# B&R Automation Studio project ABC_Pltzr
Automation Studio 4.2.2.134


## Configuration PPC70_Ver1

### Hardware
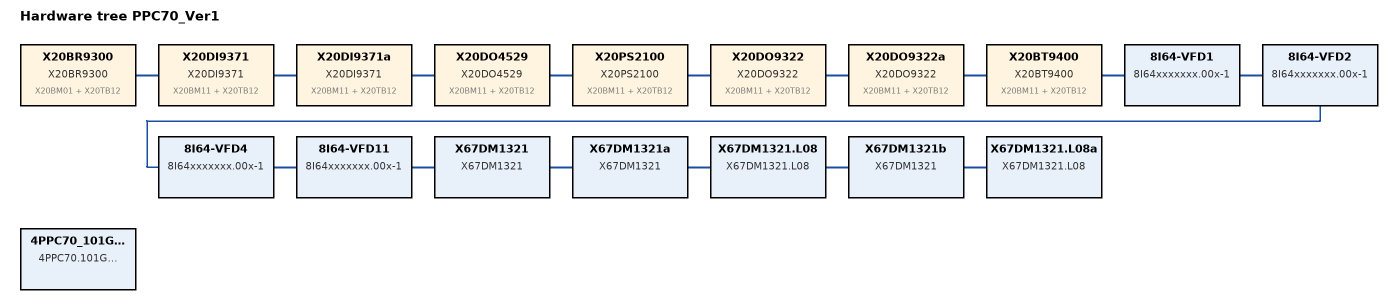
```
4PPC70_101G_20F005 : 4PPC70.101G-20F005 v1.1.0.0
  Connector IF1:
    ActivatePowerlink = 0
  Connector IF2:
    ActivateDevice = 1
    Mode = Manual
    InternetAddress = 192.168.1.100
    SubnetMask = 255.255.255.0
    InaNodeNumber = 1
    Vnc1
    VncVcObjectName1 = WSVGA
    VncKeyMappingFile1 = VC\PS2-Keyboard.dis
    VncAuthentication1 = 1
    VncPasswordViewOnly1 = v
    VncPasswordViewControl1 = eric
  Simulation = 1
  PermanentPvSize = 1000
  RemanentGlobalPvSize = 25000
  VolatileGlobalPvSize = 200000
  EnableUsbRemoteInstall = 1
  TimerDeviceType = SWIOTIMER
  Cyclic1Duration = 4000
  Cyclic1Tolerance = 4000
  Cyclic2Duration = 20000
  Cyclic2Tolerance = 20000
  Cyclic3Duration = 50000
  Cyclic3Tolerance = 50000
  Cyclic4Duration = 100000
  Cyclic4Tolerance = 100000
  Cyclic5Duration = 200000
  Cyclic5Tolerance = 200000
  Cyclic6Duration = 500000
  Cyclic6Tolerance = 500000
  Cyclic7Duration = 1000000
  Cyclic7Tolerance = 1000000
  Cyclic8Duration = 10000
  Cyclic8Tolerance = 30000000
  FtpUser1
  FtpUsername1 = abc
  FtpUserPassword1 = veVz20Da1KUF2Vww53L6omFNdzfk8lHY0HjcrjfOb/w=  // abc123
  FtpUserSalt1 = pyAcjG26
  FTPPath1 = 5
  FTPAccessRight1 = 0
  VcObjectName = WSVGA
  KeyMappingFile = VC\4PPC70_101G_20F005.dis
8I64-VFD1 : 8I64xxxxxxx.00x-1 v1.3.8.1  [X2X1 -> X20BT9400.X2X1]
  FunctionModel = Standard
  Supervision = off
  enableIOLR = off
  enableDigitalOutput = off
  DigitalOutputMode01 = actionDO
  ACC = 1
  DEC = 1
  LSP = 10
  HSP = 600
  ITH = 28
  BFR = 1
  UNS = 460
  FRS = 600
  NCR = 28
  NSP = 1750
  COS = 80
  DO = 9
  BRA = 0
  BLC = 64
  BRT = 15
  BEN = 0
  BET = 15
8I64-VFD11 : 8I64xxxxxxx.00x-1 v1.3.8.1  [X2X1 -> 8I64-VFD4.X2X2]
  FunctionModel = Standard
  Supervision = off
  enableIOLR = off
  enableDigitalOutput = off
  HSP = 600
  FTD = 600
  BFR = 1
  UNS = 460
  FRS = 600
  NCR = 15
  NSP = 1750
  COS = 80
8I64-VFD2 : 8I64xxxxxxx.00x-1 v1.3.8.1  [X2X1 -> 8I64-VFD1.X2X2]
  FunctionModel = Standard
  Supervision = off
  enableIOLR = off
  enableDigitalOutput = off
  DigitalOutputMode01 = actionDO
  DownloadParameters = yes
  ACC = 1
  DEC = 1
  BFR = 1
  UNS = 460
  FRS = 600
  NCR = 13
  NSP = 1750
  DO = 9
  BRA = 0
  BLC = 64
  BRT = 5
  BEN = 0
  BET = 5
8I64-VFD4 : 8I64xxxxxxx.00x-1 v1.3.8.1  [X2X1 -> 8I64-VFD2.X2X2]
  FunctionModel = Standard
  Supervision = off
  enableIOLR = off
  enableDigitalOutput = off
  DigitalOutputMode01 = actionDO
  DownloadParameters = yes
  ACC = 1
  DEC = 1
  HSP = 600
  ITH = 13
  FTD = 600
  BFR = 1
  UNS = 460
  FRS = 600
  NCR = 13
  NSP = 1750
  COS = 80
  DO = 9
  BRA = 0
  BLC = 64
  BRT = 5
  BEN = 0
  BET = 5
X20BM01 : X20BM01 v1.0.0.1
X20BM11 : X20BM11 v1.0.0.0  [X2X1 -> X20BM01.X2X2]
X20BM11a : X20BM11 v1.0.0.0  [X2X1 -> X20BM11.X2X2]
X20BM11b : X20BM11 v1.0.0.0  [X2X1 -> X20BM11a.X2X2]
X20BM11c : X20BM11 v1.0.0.0  [X2X1 -> X20BM11b.X2X2]
X20BM11d : X20BM11 v1.0.0.0  [X2X1 -> X20BM11c.X2X2]
X20BM11e : X20BM11 v1.0.0.0  [X2X1 -> X20BM11f.X2X2]
X20BM11f : X20BM11 v1.0.0.0  [X2X1 -> X20BM11d.X2X2]
X20BR9300 : X20BR9300 v1.0.2.6  [SS1 -> X20TB12.SS; SL -> X20BM01.SL1; X2X1 -> 4PPC70_101G_20F005.IF5]
  Supervision = off
X20BT9400 : X20BT9400 v1.0.1.3  [SS1 -> X20TB12f.SS; SL -> X20BM11e.SL1]
  Supervision = off
X20DI9371 : X20DI9371 v1.0.1.2  [SS1 -> X20TB12a.SS; SL -> X20BM11.SL1]
  Supervision = off
X20DI9371a : X20DI9371 v1.0.1.2  [SS1 -> X20TB12b.SS; SL -> X20BM11a.SL1]
  Supervision = off
  InputFilter = 100
X20DO4529 : X20DO4529 v1.0.1.2  [SS1 -> X20TB12c.SS; SL -> X20BM11b.SL1]
  Supervision = off
X20DO9322 : X20DO9322 v1.0.2.2  [SS1 -> X20TB12e.SS; SL -> X20BM11d.SL1]
  Supervision = off
X20DO9322a : X20DO9322 v1.0.2.2  [SS1 -> X20TB12g.SS; SL -> X20BM11f.SL1]
  Supervision = off
X20PS2100 : X20PS2100 v1.0.3.0  [SS1 -> X20TB12d.SS; SL -> X20BM11c.SL1]
  Supervision = off
X20TB12 : X20TB12 v1.0.0.0
X20TB12a : X20TB12 v1.0.0.0
X20TB12b : X20TB12 v1.0.0.0
X20TB12c : X20TB12 v1.0.0.0
X20TB12d : X20TB12 v1.0.0.0
X20TB12e : X20TB12 v1.0.0.0
X20TB12f : X20TB12 v1.0.0.0
X20TB12g : X20TB12 v1.0.0.0
X67DM1321 : X67DM1321 v1.1.1.0  [X2X1 -> 8I64-VFD11.X2X2]
  Supervision = off
X67DM1321.L08 : X67DM1321.L08 v1.1.2.0  [X2X1 -> X67DM1321a.X2X2]
  Supervision = off
  Direction01 = output
  Direction02 = output
  Direction03 = output
  Direction04 = output
  Direction05 = output
  Direction06 = output
  Direction07 = output
  Direction08 = output
  Direction09 = output
  Direction10 = output
  Direction11 = output
  Direction12 = output
X67DM1321.L08a : X67DM1321.L08 v1.1.2.0  [X2X1 -> X67DM1321b.X2X2]
  Supervision = off
  Direction08 = output
  Direction09 = output
X67DM1321a : X67DM1321 v1.1.1.0  [X2X1 -> X67DM1321.X2X2]
  Supervision = off
  Direction01 = output
  Direction02 = output
  Direction03 = output
  Direction04 = output
X67DM1321b : X67DM1321 v1.1.1.0  [X2X1 -> X67DM1321.L08.X2X2]
  Supervision = off
```

## Configuration testsim

CPU , AutomationRuntime D4.22, Build 4.1.2, Vc V4.22.0

### Config_1.mprecipexml - PLC1/mapp/Config_1.mprecipexml
```
Element gMpLinkMpRecipeXml (Type=mprecipexml)
```

## Logical view

Binary libraries used (declarations not repeated): AsBrStr, AsMath, AsTCP, AsUSB, Ethernet

### Program Logical/appConfigAndRecipes/appCfgRec

#### appCfgRec.c
```c
/********************************************************************
 * COPYRIGHT -- piedmont
 ********************************************************************
 * Program: cfgFS
 * File: cfgFS.c
 * Author: admin
 * Created: Jan 20, 2014
 ********************************************************************
 * Implementation of program cfgFS
 ********************************************************************/

#include <bur/plctypes.h>

#ifdef _DEFAULT_INCLUDES
 #include <AsDefault.h>
#endif

/**
 Simple logging
 Log goes to an array of PV strings > see _LOCAL STRING log[][] variable below
 Log output is visible via Automation Studio watch window
 Example of a log statement used within the code is:
 DBG("This is log example. %d ", value1);
 To complety disable logging from this source file, change next line to: #if 0
*/
#if 1
#include <../../paiComponents/bglib/bgPVLogger3.c>
#define LOG_ENTRY_COUNT 30	//max number of log entries
#define LOG_ENTRY_LENGTH  200//max length of individual log message. Longer msg are truncated
_LOCAL STRING log[LOG_ENTRY_COUNT][LOG_ENTRY_LENGTH]; //log output visible from Automation Studio!
//static bgPVLogger_typ lgr;	//PV logger object
#else
#define DBG(format, args...) ;
#define DBGINIT(args...) ;
#endif

//Support for PV serialization/deserialization
#include "../../paiComponents/bglib/bgPVSerialize.h"
#include "../appCfgRecDefault.h"
#include "../../paiComponents/paiFileService/paiPVSerDesMgr.h"
#include "../../paiComponents/paiFileService/paiFSInterface.h"
#include "../../paiComponents/paiFileService/paiFS/paiFile.h"
#include "../../paiComponents/Libraries/sprintf2/sprintf2.h"

/*
###############################################################################
PV-s
###############################################################################
*/

/*
###############################################################################
Functions
###############################################################################
*/

static void fileSetCfgFilePath(char* pCfgFilePath)
{
//Example:
//Output: pRecFilePath = "ABC/appcfg.txt"
	sprintf2(pCfgFilePath, "%s/%s", APP_DIR_NAME, APP_FILENAME_CFG);
}

/*
###############################################################################
Remanent Memory Handling
- remanent (REM) memory is battery backed SRAM
- unlike files, it has a fast, pointer based access
- in this application, it is used as a first level of storage, as follows

  working memory (DRAM) data
- valid only while CPU powered
- working memory holds all PV-s and application strucutres

Remanent memory (SRAM battery backed)
- power fail safe (only WARM restart! COLD restart deletes remanent memory)
- selected structures (eg. machine confiuration, current recipe) are copied into this area as a first level backup
- fast backup via simple memcpy

Files (CF disk)
- power fail safe and permanent
- backup requires use of FileIO access (slower, more complex)

This application combines use of the above mentioned memories.

IMPORTANT:
The REMMEM support was added before realizing that most CPU-s support only tiny (eg. 32 bytes) REM Memory areas.
As a result, the REM memory support is not really working as intended. The intended REMMEM PV-s are stored as
regular PV-s which means that these values are not preserved during power cycle.
###############################################################################
*/

static void defineFileNames()
{
	//file that holds machine configuration
	//Example: cfgFilename = "Data/appcfg.txt"
	fileSetCfgFilePath(cfgFilename);

}

/*
###############################################################################
Init, Cyclic, Exit
###############################################################################
*/
void paiPVSerDesMgrConfigure();

void _INIT appCfgRecInit( void )
{
	/* TODO: Add code here */
	DBGINIT(lgr, log, LOG_ENTRY_COUNT, LOG_ENTRY_LENGTH);

	//Define file names used for storign PV-s in this application
	defineFileNames();			//define file names used in this application

	//Configure paiSerDesMgr
	paiPVSerDesMgrConfigure();

	//TODO: gRecipe
	brsstrcpy((UDINT)gRecipe.info.name, (UDINT)"ABC");
}

void _CYCLIC appCfgRecCyclic( void )
{

	//paiFS callback execution cyclic service
	//This service executes File IO related callbacks in the context of this task
	paiFSExeCallbackCyclic(&paiFS);

	//paiSerDesMgr cyclic
	paiPVSerDesMgrCyclic(&gPVSerDesMgr);
}
//EOF
```

### notes.txt
```
9/21/2016
=========
(ProjectDate:='09/21/2016',ProjectVersion:='1.00.2',ASVersion:='AS 4.2.4',ProjectAbout:='Palletizer72',ProjectInfo:='24025',ProjectComments:='n/a')

-------- Forwarded Message --------
Subject: 	Duckhorn Wine
Date: 	Fri, 9 Sep 2016 13:25:31 +0000
From: 	David Emminger <demminger@abcpackaging.com>
To: 	Goran Bjelcevic <gbjelcevic@piedmontautomation.com>
CC: 	Eric Dederichs <edederichs@abcpackaging.com>, Greg Phelps <gphelps@piedmontautomation.com>, Kraig Downey <kdowney@abcpackaging.com>, Brittany Leslie <bleslie@abcpackaging.com>

Good morning Goran,
Duckhorn has requested a minor change to the machine HMI programming which is:

They want the fault screen to remain displayed and not automatically close when a fault is cleared. They want to manually navigate away from the fault screen.

Unhide the mute button

Change the maintenance access password to 4858418

- a logic to automaticaly switch away from the alarm screen when all alarms are cleared is removed.
Change: file: appHmiLogic.c, line: 1491
- changed the maint access password to 4858418
Change: file: paiUser.c, line: 105
- changed hide logic for safety curtains 'mute' button. Now, the button will be shown even for users that are not logged in.
Change: ladder: palletdischarge Rung: 13

5/2/2016
=======
-rectified 'no pallet reset' after executing 'Complete Pallet' manual request
-changed logic for stopping the infeed CV; instead of stopping when staging stops, the infeed CV now stops only when staging is stopped AND case is present at EE2
-changed logic for elevator when exiting pallet; instead of going to top of the pallet, now the elevator goes to the top (max elevator position)
-fixed issue with entering a case command in the layer desinger
-added support for 6th blade
-changed manual operation of the blade stops from time delayed to quick (no time delay)

4/18/2016
==========
DONE-EE2 / EE8 stop the machine row jam/incorrect count
DONE-stage at EE4
DONE-stats timer only in auto mode
-vfd fault indication in the alarm text
DONE-prevent changing counts in automatic
DONE-in automatic can't go to manual screen (put finish product button eslewhere)
-full pallet out should zero the layers
DONE ALARM INCORRECT COUNT
DONE HIDE ZERO BUTTON WHEN in AUTO
VFD BRA = OFF for VFD5 and VFD52

4/15/2016
=========
DONE: Button: load appConfig from file
VFD errors show in the alarm!
Stats counters
Case count
Pallete count
Pallete / hour
Case / min
DONE: Blade stop drawing support
DONE: Move blade stop timers to recipe
Staging cv support
Usb programming
File copy to/from to usb
Factory defaults
Retainer bar early feature
Pallet discharge interlock
Remove unused code, pages, etc
Add stop / resume to ssm.
Add single step support to ssm.

4/14/12016
=========
DONE-moved all timers to recipe
DONE-added pallet exit button (manual mode only)
DONE-added pallet finish button (auto mode only, to finish pallet and discharge)
-

4/13/2015
==========
- zero button visibility check logic (it can cause havoc is pressed when not allowed)
DONE- pallet done (in auto mode, compeltes the pallete and exits it)
 vs. run pallet out (in manual mode, exits the palette) > buttons needed
STOP BUTTON - shall stop and any time, then resume from there
PART- debounce timers for all PE-s (EE2, EE4, EE8) > recipe
DONE - product/recipe dependant settings (i.e. timers, etc)
DONE- delay front squearing action using a delay timer
DONE- pallet takeaway timer; the time required for a discharge PE to clear before the pallet are moved to discharge cv forward
- EE8 get the code for it
DONE- row forming VFD speeds and acc, table speed, acc/decl, discrage cv-s > all VDD-s shall be part of the recipe
DONE - defending fault shall be shown as the alarm!! (not low air pressure)
DONE - drop down LF key to jump to screen MANUAL
DONE - the delay time for row push shall be respected after restart following an e-stop on the last case for the row (if the e-stop tiggered just before the last estop made the row, the continue will immedialtly push the
row wo. waiting)
- Connect Alarm Ack button to the Clear VFD Fault input

3/24/2015
==========
-add alarm for elevator stop block
-add light curtain functionlity - fault and mute
-chain slack alarm recovery from stop block
-add message block stops are down

3/23/2015
=========
-added support for new HW config:
PPC70_JOB24025
-this configuration is according to the ABC JOB24025
-no palletizer dispneser is used. Instead, the pallets are build directly onto the mesh converyer
-the HW changes include:
-added 2 VFD-s VFD52 (row pusher ext) and VFD12 (pallet discharge CV)
-dropped VFD4 (row pusher) and reassinged it as VFD5 (infeed rollers)

3/22/2016
==========
-revisit and rectify recipe handling to have only a single file per recipe (i.e. layer files included in the recipe file)
-DONE-reshuffle recipe screens (i.e. recipe select, recipe create, layer create, layer view, etc)
DONE-add support for multiple blade stops
DONE-add support for pallet dispenser
-add support for infeed conveyer location (left/right) to be reflected on the configuration screen
DONE-rectify issue with the VFD-s at startup (i.e. reboot shall not be required due to incorrect configuration)
-revisti all hmi screens
-test interruptions, e-stops and power outages
-allow elevator jog when table not at grouping (recovery mode!)
-add new alarms
-pattern layer changes require reload of the pattern program to init the structures!!!

2/15/2016
==========
-revisit and rectify recipe handling to have only a single file per recipe (i.e. layer files included in the recipe file)
-reshuffle recipe screens (i.e. recipe select, recipe create, layer create, layer view, etc)
-add support for multiple blade stops
-add support for pallet dispenser
-add support for infeed conveyer location (left/right) to be reflected on the configuration screen
-rectify issue with the VFD-s at startup (i.e. reboot shall not be required due to incorrect configuration)
-revisti all hmi screens
-test interruptions, e-stops and power outages
-allow elevator jog when table not at grouping (recovery mode!)

9/10/2015
========-
-DONEadd blade stops
-DONEadd turner
-DONEestop handling
-DONEacc/dec on all drives
-DONEadd configurable number of layers

9/9/2015
=========
-add messages about zerooing machine
-add message about machine ready
-add message when auto-cycle active
-start/auto drycycle sequence

9/4/2013
========
-add number of E-Stops as an option into mach configuration
-add number of DS-s as an option into mach configuration
-add discharge light curtain to the safety logic
-remove AlwaysOnBit and TestBitx from the program when done

-add manual elevator moves to table position (use two speeds)

7/22/2015
-io
-control strructures
-alarms
-recipes
-control logic
-hmi

Subsystems:
===========
Motors ON/OFF:
-retainer bar
-row/grouping rollers
-product infeed cv
-pallet infeed chains
-pallet dispense elevator

Inverters:
-elevator
-transfer table
-row pusher
-palletizing roller cv

Machine Modes:
==============
Service (Air=NO, all motors = OFF)
Manual - HandMode (Air=YES, all motors = ON, NOT in automatic mode, manual actions)
Auto - MachineRunningAuto (automatic cycle)
DryCycle (automatic, dry cycle)
Demo (automatic, demo cycle)

Original LADDERS:
-main
-screen
-IO
-dispenser
-inserter
-bladestop1...bladestop6
-squaring
-prodset
-patterns
-picture
-caserun
-stdturner
-turntable
-servoturn
-drycycle
```

### Global.typ
```iecst
(********************************************************************
 * COPYRIGHT -- HP
 ********************************************************************
 * File: Global.typ
 * Author: goran
 * Created: January 23, 2013
 ********************************************************************
 * Global data types of project YieldPlus
 ********************************************************************)

TYPE
	applicationGlobal_enums :
		(
		APP_HWMODULE_IDXLAST := 19, (*Number of  X20 HW modules*)
		APP_CFG_BLADESTOP_MAXIDX := 5, (*Max number of blade stops*)
		APP_VFD_IDXLAST := 12 (*Max number of VFD-s*)
		);
END_TYPE
```

### Global.var
```iecst
(********************************************************************
 * COPYRIGHT -- HP
 ********************************************************************
 * File: Global.var
 * Author: goran
 * Created: January 23, 2013
 ********************************************************************
 * Global variables of project YieldPlus
 ********************************************************************)
VAR
	gProjectInfo : {REDUND_UNREPLICABLE} paiProjectInfo_typ := (ProjectDate:='09/21/2016',ProjectVersion:='1.00.2',ASVersion:='AS 4.2.4',ProjectAbout:='Palletizer72',ProjectInfo:='24025',ProjectComments:='n/a');
END_VAR
VAR RETAIN
	gREMMEMPrefix : UDINT;
	gREMMEMPostfix : UDINT;
END_VAR
```

- AlarmPopUp.fninfo (not shown)

- Arial9px.fninfo (not shown)

- Arial9pxBold.fninfo (not shown)

- Html_SDM_0.fninfo (not shown)

- Pads.fninfo (not shown)

- EditPad.tpr (not shown)

- MpNavigationPad_ver.tpr (not shown)

### brsystem.var
```iecst
(********************************************************************
 * COPYRIGHT (C) BERNECKER + RAINER, AUSTRIA, A-5142 EGGELSBERG
 ********************************************************************
 * Library: BrSystem
 * File: BrSystem.var
 * Created: 11.11.2003
 ********************************************************************
 * Constants of library BrSystem
 ********************************************************************)
VAR CONSTANT
	brSYSCONF_SET_NON_VOLATILE	: BOOL	:= TRUE;	(*set permanent value*)
	brERR_INVALID_PARAMETER	: UINT	:= 27251;		(*invalid parameter transferred*)
	brSYSCONF_SET_VOLATILE	: BOOL	:= FALSE;		(*set non-permanent value*)
	INIT_REASON_WARMSTART	: SINT	:= 1;			(*warm restart boot information*)
	INIT_REASON_COLDSTART	: SINT	:= 2;			(*cold restart boot information*)
	brERR_INVALID_DEVICE	: UINT	:= 27250;		(*battery monitoring*)
	brAUTOMATION_RUNTIME	: USINT	:= 4;			(*series recognition*)
	TARGET_LITTLE_ENDIAN	: USINT	:= 1;			(*formatSpec*)
	INIT_REASON_DOWNLOAD	: SINT	:= 3;			(*download boot information*)
	INIT_REASON_UNKNOWN	: SINT	:= -1;				(*unknown boot information*)
	brBATTERY_MISSING	: USINT	:= 3;				(*battery monitoring*)
	TARGET_BIG_ENDIAN	: USINT	:= 2;				(*formatSpec*)
	brBATTERY_NOTEST	: USINT	:= 2;				(*battery monitoring*)
	brSYSTEM_MODULE	: USINT	:= 2;					(*usage recognition*)
	brPLUGIN_MODULE	: USINT	:= 10;					(*usage recognition*)
	brLOGICSCANNER	: USINT	:= 3;					(*series recognition*)
	brBATTERY_LOW	: USINT	:= 0;					(*battery monitoring*)
	brPOWERPANEL	: USINT	:= 5;					(*series recognition*)
	brBATTERY_OK	: USINT	:= 1;					(*battery monitoring*)
	brREMOTE_IO	: USINT	:= 4;						(*usage recognition*)
	brNO_FAMILY	: USINT	:= 255;						(*series recognition*)
	brETHER_IO	: USINT	:= 6;						(*usage recognition*)
	brPRODUCT	: USINT	:= 0;						(*usage recognition*)
	brBASE_IO	: USINT	:= 3;						(*usage recognition*)
	brCAN_IO	: USINT	:= 5;						(*usage recognition*)
	brACOPOS	: USINT	:= 7;						(*usage recognition*)
	brUSRRAM	: UDINT	:= 1;						(*USRRAM memory type*)
	brSYSROM	: UDINT	:= 2;						(*SYSROM memory type*)
	brUSRROM	: UDINT	:= 3;						(*USRROM memory type*)
	brPANEL	: USINT	:= 6;							(*series recognition*)
	brADDON	: USINT	:= 7;							(*series recognition*)
	brC300	: USINT	:= 8;							(*series recognition*)
	brC200	: USINT	:= 9;							(*series recognition*)
	br2010	: USINT	:= 0;							(*series recognition*)
	br2005	: USINT	:= 1;							(*series recognition*)
	br2003	: USINT	:= 2;							(*series recognition*)
	brDRAM	: UDINT	:= 0;							(*DRAM memory type*)
	brKEY	: USINT	:= 8;							(*usage recognition*)
	brCPU	: USINT	:= 1;							(*usage recognition*)
	brPP	: USINT	:= 255;							(*usage recognition*)
	brX2X	: USINT	:= 10;							(*series recognition*)
END_VAR
```

### dvframe.var
```iecst
(********************************************************************
 * COPYRIGHT (C) BERNECKER + RAINER, AUSTRIA, A-5142 EGGELSBERG
 ********************************************************************
 * Library:    DVFrame
 * File:            DVFrame.var
 * Created:         11.11.2003
 ********************************************************************
 * Constants of library DVFrame
 ********************************************************************)
VAR CONSTANT
	frmERR_IOCTL_NOTSUPPORTED	: UINT	:= 8257;	(*command not supported by driver (hardware)*)
	frmERR_DEVICEDESCRIPTION	: UINT	:= 8252;	(*device not found*)
	frmERR_FUB_ENABLE_FALSE	: UINT	:= 65534;
	frmERR_TRANSMITOVERRUN	: UINT	:= 8078;		(*send buffer waiting queue full*)
	frmERR_MODEDESCRIPTION	: UINT	:= 8253;		(*syntax error in mode parameter string, or mode parameter not supported by the specified device*)
	frmERR_IOCTL_NOTVALID	: UINT	:= 8073;		(*invalid I/O control code*)
	frmERR_INVALIDBUFFER	: UINT	:= 8072;		(*invalid buffer rejected*)
	ARG_EVSEND_TASKIDENT	: UDINT	:= 14;
	ARG_EVSEND_TASKEVENT	: UDINT	:= 18;
	frmERR_NORESOURCES	: UINT	:= 8258;			(*required resource not available (memory, OS object, etc.)*)
	frmERR_INPUTERROR	: UINT	:= 8079;			(*frame buffer with defective character*)
	frmERR_NOTOPENED	: UINT	:= 8251;			(*device not open*)
	MISC_RECEIVE_ALL	: UDINT	:= 2;
	frmERR_PA_DB_SB	: UINT	:= 8256;				(*/PA, /DB, /SB must always be specified together*)
	frmERR_NOBUFFER	: UINT	:= 8071;				(*no buffer available in the send buffer manager*)
	ARG_TXPVPOLLADR	: UDINT	:= 17;
	frmERR_NOINPUT	: UINT	:= 60;					(*no message received*)
	frmERR_MAXOPEN	: UINT	:= 8254;				(*too many devices opened at once*)
	ARG_PVPOLLADR	: UDINT	:= 15;
	frmERR_OK	: UINT	:= 0;
	ARG_MISC	: UDINT	:= 16;
	ARG_BAUD	: UDINT	:= 0;
END_VAR
```

- vssver.scc (binary file, 48 bytes)
### MpFile.typ
```iecst
TYPE
	MpFileManagerUIItemType : 	STRUCT
		Name : STRING[255]; (*Filename / Folder name*)
		Size : UDINT; (*File size [bytes]*)
		LastModified : DATE_AND_TIME; (*Date when this file/folder was last modified*)
		ItemType : MpFileManagerUIItemTypeEnum; (*File type (.csv, .jpg, etc.)*)
		IsSelected : BOOL; (*Indicates that a file/folder is selected*)
		IsFolder : BOOL; (*Indicates that the element is a folder*)
	END_STRUCT;
	MpFileManagerUIItemTypeEnum :
		(
		mpFILE_ITEM_TYPE_NONE := 0, (*No type defined*)
		mpFILE_ITEM_TYPE_FOLDER := 1, (*Indicates that the element is a folder*)
		mpFILE_ITEM_TYPE_FILE := 2, (*Indicates that the element is a file*)
		mpFILE_ITEM_TYPE_TXT := 3, (*Indicates that the element is a text file*)
		mpFILE_ITEM_TYPE_HTML := 4, (*Indicates that the element is an HTML file*)
		mpFILE_ITEM_TYPE_DOC := 5, (*Indicates that the element is a Word file (.doc) *)
		mpFILE_ITEM_TYPE_XLS := 6, (*Indicates that the element is an Excel file (.xls)*)
		mpFILE_ITEM_TYPE_XML := 7, (*Indicates that the element is an XML file (.xml)*)
		mpFILE_ITEM_TYPE_CSV := 8, (*Indicates that the element is an CSV file (.csv)*)
		mpFILE_ITEM_TYPE_JPG := 9, (*Indicates that the element is an image file (.jpg)*)
		mpFILE_ITEM_TYPE_BMP := 10, (*Indicates that the element is an image file (.bmp)*)
		mpFILE_ITEM_TYPE_USER1 := 89, (*Indicates that the element is an user predefined type 1*)
		mpFILE_ITEM_TYPE_USER2 := 90, (*Indicates that the element is an user predefined type 2*)
		mpFILE_ITEM_TYPE_USER3 := 91, (*Indicates that the element is an user predefined type 3*)
		mpFILE_ITEM_TYPE_USER4 := 92, (*Indicates that the element is an user predefined type 4*)
		mpFILE_ITEM_TYPE_USER5 := 93, (*Indicates that the element is an user predefined type 5*)
		mpFILE_ITEM_TYPE_USER6 := 94, (*Indicates that the element is an user predefined type 6*)
		mpFILE_ITEM_TYPE_USER7 := 95, (*Indicates that the element is an user predefined type 7*)
		mpFILE_ITEM_TYPE_USER8 := 96, (*Indicates that the element is an user predefined type 8*)
		mpFILE_ITEM_TYPE_USER9 := 97, (*Indicates that the element is an user predefined type 9*)
		mpFILE_ITEM_TYPE_USER10 := 98, (*Indicates that the element is an user predefined type 10*)
		mpFILE_ITEM_TYPE_UNKNOWN := 99 (*Indicates that the file type is unknown*)
		);
	MpFileManagerUISortOrderEnum :
		(
		mpFILE_SORT_BY_NAME_ASC := 0, (*Sorts in ascending (alphabetic) order*)
		mpFILE_SORT_BY_NAME_DESC := 1, (*Sorts in descending (alphabetic) order*)
		mpFILE_SORT_BY_SIZE_ASC := 2, (*Sorts in ascending order by file size*)
		mpFILE_SORT_BY_SIZE_DES := 3, (*Sorts in descending order by file size*)
		mpFILE_SORT_BY_MOD_TIME_ASC := 4, (*Sorts in ascending order by date last modified*)
		mpFILE_SORT_BY_MOD_TIME_DESC := 5 (*Sorts in descending order by date last modified*)
		);
	MpFileManagerUIMessageEnum :
		(
		mpFILE_MSG_OK := 0, (*Dialog box for requesting confirmation of input*)
		mpFILE_MSG_CONFIRM_DELETE := 1, (*Dialog box for requesting confirmation of deletion*)
		mpFILE_MSG_CONFIRM_OVERWRITE := 2, (*Dialog box for requesting confirmation of overwriting*)
		mpFILE_MSG_BUSY := 3 (*Dialog box for requesting confirmation of busy UI*)
		);
	MpFileDiagType : 	STRUCT
		StatusID : MpFileStatusIDType; (*StatusID diagnostic structure*)
	END_STRUCT;
	MpFileStatusIDType : 	STRUCT
		ID : MpFileErrorEnum; (*Error code for mapp component*)
		Severity : MpComSeveritiesEnum; (*Describes the type of information supplied by the status ID (success, information, warning, error)*)
		Code : UINT; (*Code for the status ID. This error number can be used to search for additional information in the help system.*)
	END_STRUCT;
	MpFileInfoType : 	STRUCT
		Diag : MpFileDiagType; (*Diagnostic structure for the status ID*)
	END_STRUCT;
	MpFileManagerUIStatusEnum :
		(
		mpFILE_UI_STATUS_IDLE := 0, (*Indicates that no process is currently active*)
		mpFILE_UI_STATUS_REFRESH := 1, (*Updating elements*)
		mpFILE_UI_STATUS_CHANGE_PAGE := 2, (*Page change active*)
		mpFILE_UI_STATUS_CHANGE_DIR := 3, (*Folder change active*)
		mpFILE_UI_STATUS_CHANGE_DEVICE := 4, (*File Device Change active*)
		mpFILE_UI_STATUS_CREATE := 5, (*Creating a file/folder active*)
		mpFILE_UI_STATUS_RENAME := 6, (*Renaming a file/folder active*)
		mpFILE_UI_STATUS_DELETE := 7, (*Deleting a file/folder active*)
		mpFILE_UI_STATUS_COPY := 8, (*Copying a file/folder active*)
		mpFILE_UI_STATUS_CUT := 9, (*Cutting a file/folder active*)
		mpFILE_UI_STATUS_PASTE := 10, (*Pasting a file/folder active*)
		mpFILE_UI_STATUS_SORT := 11, (*Sorting files/folders in specified sort order*)
		mpFILE_UI_STATUS_ERROR := 99 (*The last operation generated an error*)
		);
	MpFileManagerUISetupType : 	STRUCT
		FileListSize : UINT := 10; (*Number of files to be displayed on one page of the list in the HMI application*)
		FileListScrollWindow : USINT := 1; (*Determines how many entries from the list are displayed in advance when scrolling up and down*)
	END_STRUCT;
	MpFileManagerUIConnectType : 	STRUCT
		Status : MpFileManagerUIStatusEnum; (*Current operation*)
		DeviceList : MpFileManagerUIDeviceListType; (*List of data storage media (file devices) accessible by the file manager*)
		File : MpFileManagerUIFileType; (*Contains the file list as well as additional information about files,folders and possible commands*)
		MessageBox : MpFileManagerUIMessageBoxType; (*Controls dialog boxes*)
		DefaultLayerStatus : UINT; (*Status DP for the default layer of the visu page where the file manager is being displayed*)
	END_STRUCT;
	MpFileManagerUIMessageBoxType : 	STRUCT
		LayerStatus : UINT; (*Visibility of the dialog box*)
		Type : MpFileManagerUIMessageEnum; (*Type of dialog box*)
		ErrorNumber : UINT; (*Current error number to be displayed*)
		Confirm : BOOL; (*Confirms the operation*)
		Cancel : BOOL; (*Cancels the operation*)
	END_STRUCT;
	MpFileManagerUIPathInfoType : 	STRUCT
		CurrentDir : STRING[255]; (*Current folder name*)
		FileCount : UDINT; (*Number of files in the current folder*)
		FolderCount : UDINT; (*Number of subfolders in the current folder*)
	END_STRUCT;
	MpFileManagerUIFileType : 	STRUCT
		List : MpFileManagerUIFileListType; (*List of all folders and files under the current path, as well as the navigation of the list*)
		Filter : STRING[255]; (*Filter used to sort the files*) (* *) (*#CMD#OPT#;*)
		SortOrder : MpFileManagerUISortOrderEnum; (*Responsible for the order of files in the list*)
		Refresh : BOOL; (*Updates the file list in the current folder*)
		PathInfo : MpFileManagerUIPathInfoType; (*Information about the current path*)
		EnterFolder : BOOL; (*Navigates one folder down*)
		FolderUp : BOOL; (*Navigates one folder up*)
		MultiSelect : BOOL; (*Allows the selection of multiple elements at the same time*)
		Delete : BOOL; (*Deletes a file or folder*)
		Copy : BOOL; (*Copying a file/folder*)
		Cut : BOOL; (*Cuts a file or folder*)
		Paste : BOOL; (*Pastes a file or folder*)
		NewName : STRING[255]; (*The new name of a file or folder when using the "Rename" or "CreateFolder" command*)
		Rename : BOOL; (*Renames a file or folder*)
		CreateFolder : BOOL; (*Creates a folder*)
	END_STRUCT;
	MpFileManagerUIFileListType : 	STRUCT
		Items : ARRAY[0..49]OF MpFileManagerUIItemType; (*List of all files and folders under the current path*)
		PageUp : BOOL; (*Jumps to the start of the current page and then scrolls up one page at a time*)
		StepUp : BOOL; (*Selects the previous entry in the list*)
		PageDown : BOOL; (*Jumps to the end of the current page and then scrolls down one page at a time*)
		StepDown : BOOL; (*Selects the next entry in the list*)
		RangeStart : REAL; (*Shows a bar indicating which part of the list is currently being displayed-Start [%]*)
		RangeEnd : REAL; (*Shows a bar indicating which part of the list is currently being displayed-End [%]*)
	END_STRUCT;
	MpFileManagerUIDeviceListType : 	STRUCT
		DeviceNames : ARRAY[0..9]OF STRING[50]; (*List of all available data storage media*)
		SelectedIndex : UINT; (*Index of the entry currently selected in the list*)
	END_STRUCT;
END_TYPE
```

- vssver.scc (binary file, 48 bytes)
- Program Logical/MachineControl/animation (IEC) (no source held here)

### Program Logical/MachineControl/appHmi

#### appHmiLogic.c
```c
/********************************************************************
 * COPYRIGHT -- pai
 ********************************************************************
 * Program: hmilogic
 * File: hmilogic.c
 * Author: goran
 * Created: August 28, 2013
 ********************************************************************
 * Implementation of program hmilogic
 ********************************************************************/

#include <bur/plctypes.h>

#ifdef _DEFAULT_INCLUDES
	#include <AsDefault.h>
#endif

#include "../../paiComponents/paiHmi/paiHmiParamList.h"
#include "../../paiComponents/paiHmi/paiHmiPageChange.h"
#include "../../paiComponents/paiHmi/paiHmiAlert.h"
#include "../../paiComponents/bglib/bgBitUtilities.h"

/*
###############################################################################
Utilities
###############################################################################
*/

/**
Screen ID-s must match AutomationStudio's  VisualComponents Page Numbers!!!!!
NOTE: not all screen must have logic support written in this file! Actually,
less logic here and using more VC features is a prefered approach to
implement VC HMI apps.
*/
enum{
	SID_Init = 0,
	SID_Main = 10,
	SID_Main_Monitor = 11,
	SID_Settings_System = 60,
	SID_Settings_Timers = 61,
	SID_Settings_VFDs = 62,
	SID_Settings_Options = 63,
	SID_Settings_MachCfg = 65,
	SID_Recipe_LayerDesign = 44,
	SID_Recipe_LayerPreview = 41,
	SID_Recipe_PalletSelect = 46,
	SID_Recipe_PalletConfig = 45,
	SID_Recipe_PalletTimers = 47,
	SID_Recipe_PalletVFDs = 48,
	SID_Diag_Alarms = 81,
	SID_System_Files = 103,
	SID_Manual = 82,
	SID_Manual2 = 87,

	SID_MAX  /*always last!!!*/
}APPSCREENIDS;

/**
Application specific HMI dialogs must be unique. Always to in pair (accept,reject, etc)
*/
enum{
	DLG_Ok = 10,
	DLG_Cancel,
	DLG_DeleteL1FilenameOK = 20,
	DLG_DeleteL1FilenameCancel,
	DLG_SaveAppConfigOK = 30,
	DLG_SaveAppConfigCancel,
	DLG_SavePalletRecipeOK = 40,
	DLG_SavePalletRecipeCancel,

}APPHMIDIALOGIDS;

/*
###############################################################################
Parameter view/edit tables
###############################################################################
*/

/*
###############################################################################
Parameter view/edit tables
###############################################################################
*/
static void hmiTableRecipeTimers()
{
	//configApp_typ* pAppCfg = &gConfigApp;
	palleteCfgSettings_typ* pAppCfg = &gPallete.palCfg.palSettings;

	//	DINT decFormat_None = -2; //no dec places
	//	DINT decFormat_0 = -1;    //1 dec place
	DINT decFormat_00 = 0;    //default (2) dec places as set in the control
	//	DINT decFormat_000 = 1;    //3 dec places

	//scaling
	//y=kx+n where: y=HMI value, x=PLC value
	REAL k_factor = 1.0;
	REAL n_factor = 0.0;
	//	UINT valtypeUDINT = 0;//UDINT
	UINT valtypeREAL = 1;//REAL

	hmiParamListTableEntryFirst(&gHmiParamTable, "Pallet Timers");

//#if 0
	hmiParamListTableAddEntryNext(&gHmiParamTable,
		(UDINT)&pAppCfg->timers.dlyTableLayerRdyToElevMove , "TableReadyToElevatorMove",
		1.0, 0.1, 5.0,
		decFormat_00, k_factor, n_factor, valtypeREAL, "Delay time from Table Layer Ready to Elevator Move [sec].");

	hmiParamListTableAddEntryNext(&gHmiParamTable,
		(UDINT)&pAppCfg->timers.dlyTableAtPalleteToRetBar , "DelayRetainerBarMoveDown",
		1.0, 0.1, 5.0,
		decFormat_00, k_factor, n_factor, valtypeREAL, "Delay time from Table at Pallet to Retainer Bar move down to Squaring [sec].");

	hmiParamListTableAddEntryNext(&gHmiParamTable,
		(UDINT)&pAppCfg->timers.onDlyPRRetBarDown , "DelayRetainerBarIsDown",
		0.05, 0.00, 1.0,
		decFormat_00, k_factor, n_factor, valtypeREAL, "On delay for Retainer Bar Down Prox sensor [sec]. Higher value > layer edge gets positioned deeper inside the pallete.");

	hmiParamListTableAddEntryNext(&gHmiParamTable,
		(UDINT)&pAppCfg->timers.onDlyEEPallete , "onDelayEE1Pallet",
		0.05, 0.00, 1.0,
		decFormat_00, k_factor, n_factor, valtypeREAL, "On delay for Pallet Sensor EE1[sec]. Longer delay results in table getting closer to the pallete when dropping a layer. DANGER: Setting this time too long may cause mechanical colision!");

	hmiParamListTableAddEntryNext(&gHmiParamTable,
		(UDINT)&pAppCfg->timers.offDlyEEPallete , "offDelayEE1Pallet",
		0.05, 0.00, 3.0,
		decFormat_00, k_factor, n_factor, valtypeREAL, "Off delay for Pallet Sensor EE1[sec].");

	hmiParamListTableAddEntryNext(&gHmiParamTable,
		(UDINT)&pAppCfg->timers.onDlyPalleteDischargeEE16 , "onDelayPalleteDischargeEE16",
		0.05, 0.00, 3.0,
		decFormat_00, k_factor, n_factor, valtypeREAL, "On delay for Pallet Discharge Sensor EE16[sec]. Longer delay results in pallete getting futher on the discharge CV. DANGER: Setting this time too long may cause pallete tip over!");

	hmiParamListTableAddEntryNext(&gHmiParamTable,
		(UDINT)&pAppCfg->timers.onTmCaseTurner , "onTimeCaseTurner",
		1.0, 0.1, 5.0,
		decFormat_00, k_factor, n_factor, valtypeREAL, "On Time for case turner[sec].");

	hmiParamListTableAddEntryNext(&gHmiParamTable,
		(UDINT)&pAppCfg->timers.dlyRowDoneToRowPush , "DelayForRowDoneToRowPush",
		1.0, 0.1, 5.0,
		decFormat_00, k_factor, n_factor, valtypeREAL, "Delay time from row forming conmplete signal to push the row to the table [sec].");

	hmiParamListTableAddEntryNext(&gHmiParamTable,
		(UDINT)&pAppCfg->timers.dlyLastCaseToRowCVStop , "DelayLastCaseToRowConvStop",
		1.0, 0.1, 5.0,
		decFormat_00, k_factor, n_factor, valtypeREAL, "Delay from the moment the last case for a row passes by EE4 until a row forming CV is stopped[sec].");

	hmiParamListTableAddEntryNext(&gHmiParamTable,
		(UDINT)&pAppCfg->timers.dlyPusherAtElevatorToRetract , "DelayPusherAtElevatorReturnToHome",
		1.0, 0.1, 5.0,
		decFormat_00, k_factor, n_factor, valtypeREAL, "Delay from the moment row pusher gets to the elevator before a reverse motion is started to retract row pusher back to home[sec].");

	hmiParamListTableAddEntryNext(&gHmiParamTable,
		(UDINT)&pAppCfg->timers.dlyTableAtPalleteToRetBar , "DelayTableFwdToRetainerBarDown",
		1.0, 0.0, 5.0,
		decFormat_00, k_factor, n_factor, valtypeREAL, "Delay from a moment the table starts moving towards the pallet top and before a retainter bar starts moving down[sec]. NOTE: Setting this value too short may cause a collision.");

	hmiParamListTableAddEntryNext(&gHmiParamTable,
		(UDINT)&pAppCfg->timers.onDlyTableToGrouping , "DelayTableToGrouping",
		0.0, 0.0, 2.0,
		decFormat_00, k_factor, n_factor, valtypeREAL, "Delay from a moment the layer is dropped onto the top of the pallet and before table starts moving towards the grouping[sec].");

	hmiParamListTableAddEntryNext(&gHmiParamTable,
		(UDINT)&pAppCfg->timers.JamAlarmTmAtInfeedEE2 , "JamAlarmTimeAtCaseInfeedEE2",
		4.0, 1.0, 20.0,
		decFormat_00, k_factor, n_factor, valtypeREAL, "Maximum time allowed to block the EE2 Case Infeed PE before a jam alarm is generated [sec].");

	hmiParamListTableAddEntryNext(&gHmiParamTable,
		(UDINT)&pAppCfg->timers.JamAlarmTmAtRowToLongEE8 , "JamAlarmTimeAtRowToLongEE8",
		4.0, 1.0, 20.0,
		decFormat_00, k_factor, n_factor, valtypeREAL, "Maximum time allowed to block the EE8 Row Too Long PE before an alarm is generated [sec].");

	hmiParamListTableAddEntryNext(&gHmiParamTable,
		(UDINT)&pAppCfg->timers.JamAlarmTmRowForming , "JamAlarmTimeAtRowForming",
		4.0, 1.0, 20.0,
		decFormat_00, k_factor, n_factor, valtypeREAL, "Maximum time allowed for a case to travel between EE2 (Case Infeed PE) and EE8 (Row Too Long PE) before an alarm is generated [sec].");

	hmiParamListTableAddEntryNext(&gHmiParamTable,
		(UDINT)&pAppCfg->timers.infeedCVIdleTime , "InfeedCVIdleTime",
		30.0, 10.0, 600.0,
		decFormat_00, k_factor, n_factor, valtypeREAL, "Maximum idle time for infeed CV-s before they get turned off[sec].");

	hmiParamListTableAddEntryNext(&gHmiParamTable,
		(UDINT)&pAppCfg->timers.palletExitAlarmTm , "PalletExitAlarmTime",
		15.0, 5.0, 60.0,
		decFormat_00, k_factor, n_factor, valtypeREAL, "Maximum time allowed for a pallet to exit the machine (i.e. activate EE16) [sec].");
//#endif

	hmiParamListTableAddEntryNext(&gHmiParamTable,
		(UDINT)&pAppCfg->timers.EE2OnDebounce , "EE2OnDebounce",
		0.0, 0.0, 0.5,
		decFormat_00, k_factor, n_factor, valtypeREAL, "EE2 (Infeed) On debounce time[sec].");

	hmiParamListTableAddEntryNext(&gHmiParamTable,
		(UDINT)&pAppCfg->timers.EE2OfDebounce , "EE2OffDebounce",
		0.0, 0.0, 0.5,
		decFormat_00, k_factor, n_factor, valtypeREAL, "EE2 (Infeed) Off debounce time[sec].");

	hmiParamListTableAddEntryNext(&gHmiParamTable,
		(UDINT)&pAppCfg->timers.EE4OnDebounce , "EE4OnDebounce",
		0.0, 0.0, 0.5,
		decFormat_00, k_factor, n_factor, valtypeREAL, "EE4 (Stage CV PE) On debounce time[sec].");

	hmiParamListTableAddEntryNext(&gHmiParamTable,
		(UDINT)&pAppCfg->timers.EE4OfDebounce , "EE4OffDebounce",
		0.0, 0.0, 0.5,
		decFormat_00, k_factor, n_factor, valtypeREAL, "EE4 (Stage CV PE) Off debounce time[sec].");

	hmiParamListTableAddEntryNext(&gHmiParamTable,
		(UDINT)&pAppCfg->timers.EE8OnDebounce , "EE8OnDebounce",
		0.0, 0.0, 0.5,
		decFormat_00, k_factor, n_factor, valtypeREAL, "EE8 (Row To Long) On debounce time[sec].");

	hmiParamListTableAddEntryNext(&gHmiParamTable,
		(UDINT)&pAppCfg->timers.EE8OfDebounce , "EE8OffDebounce",
		0.0, 0.0, 0.5,
		decFormat_00, k_factor, n_factor, valtypeREAL, "EE8 (Row To Long) Off debounce time[sec].");

	hmiParamListTableAddEntryNext(&gHmiParamTable,
		(UDINT)&pAppCfg->timers.EE16OfDebounce , "EE16OffDebounce",
		5.0, 0.0, 60.0,
		decFormat_00, k_factor, n_factor, valtypeREAL, "EE16 (Pallete Discharge Sensor) Off debounce time[sec]. Longer time prevents to quick exiting of a pallete from the staging CV to discharge CV after EE16 gets unblocked.");

	hmiParamListTableAddEntryNext(&gHmiParamTable,
		(UDINT)&pAppCfg->timers.onDlyFrontSquaring , "FrontSquaringOnDelay",
		0.0, 0.0, 3.0,
		decFormat_00, k_factor, n_factor, valtypeREAL, "Front Squaring On Delay[sec]. Allows for a delayed action of the front squaring bar to prevent product pushing.");

	if(gConfigApp.system.bladeStopCount >= 1){
		hmiParamListTableAddEntryNext(&gHmiParamTable,
			(UDINT)&pAppCfg->timers.bladeStopOnDly1 , "Blade1TurnOnDelay",
			1.0, 0.0, 10.0,
			decFormat_00, k_factor, n_factor, valtypeREAL, "Blade 1 turn-on delay. Delayed turn-on when executing pattern program is required so that the blade does not block an incorrect case [sec].");
	}

	if(gConfigApp.system.bladeStopCount >= 2){
		hmiParamListTableAddEntryNext(&gHmiParamTable,
			(UDINT)&pAppCfg->timers.bladeStopOnDly2 , "Blade2TurnOnDelay",
			2.0, 0.0, 10.0,
			decFormat_00, k_factor, n_factor, valtypeREAL, "Blade 2 turn-on delay. Delayed turn-on when executing pattern program is required so that the blade does not block an incorrect case [sec]");
	}

	if(gConfigApp.system.bladeStopCount >= 3){
		hmiParamListTableAddEntryNext(&gHmiParamTable,
			(UDINT)&pAppCfg->timers.bladeStopOnDly3 , "Blade3TurnOnDelay",
			3.0, 0.0, 10.0,
			decFormat_00, k_factor, n_factor, valtypeREAL, "Blade 3 turn-on delay. Delayed turn-on when executing pattern program is required so that the blade does not block an incorrect case [sec]");
	}

	if(gConfigApp.system.bladeStopCount >= 4){
		hmiParamListTableAddEntryNext(&gHmiParamTable,
			(UDINT)&pAppCfg->timers.bladeStopOnDly4 , "Blade4TurnOnDelay",
			4.0, 0.0, 10.0,
			decFormat_00, k_factor, n_factor, valtypeREAL, "Blade 4 turn-on delay. Delayed turn-on when executing pattern program is required so that the blade does not block an incorrect case [sec]");
	}

	if(gConfigApp.system.bladeStopCount >= 5){
		hmiParamListTableAddEntryNext(&gHmiParamTable,
			(UDINT)&pAppCfg->timers.bladeStopOnDly5 , "Blade5TurnOnDelay",
			5.0, 0.0, 10.0,
			decFormat_00, k_factor, n_factor, valtypeREAL, "Blade 5 turn-on delay. Delayed turn-on when executing pattern program is required so that the blade does not block an incorrect case [sec]");
	}

	hmiParamListTableEntryLast(&gHmiParamTable);

}

static void hmiTableOptions()
{
	configApp_typ* pAppCfg = &gConfigApp;

	DINT decFormat_None = -2; //no dec places
//	DINT decFormat_0 = -1;    //1 dec place
	DINT decFormat_00 = 0;    //default (2) dec places as set in the control
//	DINT decFormat_000 = 1;    //3 dec places

	//scaling
	//y=kx+n where: y=HMI value, x=PLC value
	REAL k_factor = 1.0;
	REAL n_factor = 0.0;
	UINT valtypeUDINT = 0;//UDINT
	UINT valtypeREAL = 1;//REAL

	hmiParamListTableEntryFirst(&gHmiParamTable, "Options");

	hmiParamListTableAddEntryNext(&gHmiParamTable,
		(UDINT)&pAppCfg->options.dryCycleCaseCount, "DryCycleCaseCount",
		5.0, 1.0, 5.0,
		decFormat_None, k_factor, n_factor, valtypeUDINT, "Number of cases per row during DryCycle.");

	hmiParamListTableAddEntryNext(&gHmiParamTable,
		(UDINT)&pAppCfg->options.dryCycleRowCount, "DryCycleRowCount",
		4.0, 1.0, 4.0,
		decFormat_None, k_factor, n_factor, valtypeUDINT, "Number of rows per layer during DryCycle.");

	hmiParamListTableAddEntryNext(&gHmiParamTable,
		(UDINT)&pAppCfg->options.dryCycleLayerCount, "DryCycleLayerCount",
		3.0, 1.0, 6.0,
		decFormat_None, k_factor, n_factor, valtypeUDINT, "Number of layers on the pallet during DryCycle.");

	hmiParamListTableAddEntryNext(&gHmiParamTable,
		(UDINT)&pAppCfg->options.tmDryCycleElevatorUp, "DryCycleElevatorUp Time",
		3.0, 1.0, 5.0,
		decFormat_00, k_factor, n_factor, valtypeREAL, "DryCycle simulation timer for simulating layers [sec].");

	hmiParamListTableAddEntryNext(&gHmiParamTable,
		(UDINT)&pAppCfg->options.tmDryCycleCaseTime , "DryCycleCase Time",
		2.0, 1.0, 5.0,
		decFormat_00, k_factor, n_factor, valtypeREAL, "DryCycle simulation time for simulating loading a single case [sec].");

	hmiParamListTableAddEntryNext(&gHmiParamTable,
		(UDINT)&pAppCfg->options.tmDryCycleLayerZeroOffset , "DryCycleLayer0Offset",
		2.0, 1.0, 5.0,
		decFormat_00, k_factor, n_factor, valtypeREAL, "DryCycle layer 0 offset time. Alows elevator position control for the layer 0. [sec].");

	hmiParamListTableAddEntryNext(&gHmiParamTable,
		(UDINT)&pAppCfg->options.dryCycleLayerDonePause , "DryCyclePause",
		0.0, 0.0, 1.0,
		decFormat_None, k_factor, n_factor, valtypeUDINT, "0-continues DryCycle operation, 1-pause after layer completion during DryCycle.");

	hmiParamListTableEntryLast(&gHmiParamTable);

}

static void hmiTableRecipeVFDs()
{
	//configApp_typ* pAppCfg = &gConfigApp;
	palleteCfgSettings_typ* pAppCfg = &gPallete.palCfg.palSettings;

	DINT decFormat_None = -2; //no dec places
	//DINT decFormat_0 = -1;    //1 dec place
	//DINT decFormat_00 = 0;    //default (2) dec places as set in the control
	//	DINT decFormat_000 = 1;    //3 dec places

	//scaling
	//y=kx+n where: y=HMI value, x=PLC value
	REAL k_factor = 1.0;
	REAL n_factor = 0.0;
	UINT valtypeUDINT = 0;//UDINT
	//	UINT valtypeREAL = 1;//REAL

	hmiParamListTableEntryFirst(&gHmiParamTable, "Pallet VFD Settings");

	hmiParamListTableAddEntryNext(&gHmiParamTable,
		(UDINT)&pAppCfg->vfd[1].velocity_rpm, "VelocityVFD1",
		300.0, 0.0, 2700.0,
		decFormat_None, k_factor, n_factor, valtypeUDINT, "VFD1(Elevator) Velocity [rpm]");

	hmiParamListTableAddEntryNext(&gHmiParamTable,
		(UDINT)&pAppCfg->vfd[1].velocitySlow_rpm, "VelocityVFD1Slow",
		150.0, 0.0, 2700.0,
		decFormat_None, k_factor, n_factor, valtypeUDINT, "VFD1(Elevator) Slow Velocity. Used when approaching home position [rpm]");

	hmiParamListTableAddEntryNext(&gHmiParamTable,
		(UDINT)&pAppCfg->vfd[2].velocity_rpm, "VelocityVFD2",
		300.0, 0.0, 2700.0,
		decFormat_None, k_factor, n_factor, valtypeUDINT, "VFD2(Table) Velocity [rpm]");
#if 0
	hmiParamListTableAddEntryNext(&gHmiParamTable,
		(UDINT)&pAppCfg->vfd[4].velocity_rpm, "VelocityVFD4",
		300.0, 0.0, 2700.0,
		decFormat_None, k_factor, n_factor, valtypeUDINT, "VFD4(Row Pusher) Velocity [rpm]");
#endif

	hmiParamListTableAddEntryNext(&gHmiParamTable,
		(UDINT)&pAppCfg->vfd[5].velocity_rpm, "VelocityVFD5",
		300.0, 0.0, 2700.0,
		decFormat_None, k_factor, n_factor, valtypeUDINT, "VFD5 Row Forming Rollers Velocity [rpm]");

	hmiParamListTableAddEntryNext(&gHmiParamTable,
		(UDINT)&pAppCfg->vfd[6].velocity_rpm, "VelocityVFD52",
		300.0, 0.0, 2700.0,
		decFormat_None, k_factor, n_factor, valtypeUDINT, "VFD52 Row Forming Rollers 2 Velocity [rpm]");

	hmiParamListTableAddEntryNext(&gHmiParamTable,
		(UDINT)&pAppCfg->vfd[11].velocity_rpm, "VelocityVFD11",
		300.0, 0.0, 2700.0,
		decFormat_None, k_factor, n_factor, valtypeUDINT, "VFD11 (Pallet Forming Mesh CV) Velocity [rpm]");

	hmiParamListTableAddEntryNext(&gHmiParamTable,
		(UDINT)&pAppCfg->vfd[12].velocity_rpm, "VelocityVFD12",
		300.0, 0.0, 2700.0,
		decFormat_None, k_factor, n_factor, valtypeUDINT, "VFD12(Pallet Discharge Mesh CV) Velocity [rpm]");

	//Acceleration
	hmiParamListTableAddEntryNext(&gHmiParamTable,
		(UDINT)&pAppCfg->vfd[1].acc, "AccelVFD1",
		1.0, 1.0, 10.0,
		decFormat_None, k_factor, n_factor, valtypeUDINT, "VFD1(Elevator) Acceleration [0.1 sec]");

	hmiParamListTableAddEntryNext(&gHmiParamTable,
		(UDINT)&pAppCfg->vfd[2].acc, "AccelVFD2",
		1.0, 1.0, 20.0,
		decFormat_None, k_factor, n_factor, valtypeUDINT, "VFD2(Table) Acceleration [0.1 sec]");

	hmiParamListTableAddEntryNext(&gHmiParamTable,
		(UDINT)&pAppCfg->vfd[5].acc, "AccelVFD5",
		1.0, 1.0, 20.0,
		decFormat_None, k_factor, n_factor, valtypeUDINT, "VFD5(Row Forming Rollers) Acceleration [0.1 sec]");

	hmiParamListTableAddEntryNext(&gHmiParamTable,
		(UDINT)&pAppCfg->vfd[6].acc, "AccelVFD52",
		1.0, 1.0, 20.0,
		decFormat_None, k_factor, n_factor, valtypeUDINT, "VFD52(Row Forming Rollers 2) Acceleration [0.1 sec]");

	hmiParamListTableAddEntryNext(&gHmiParamTable,
		(UDINT)&pAppCfg->vfd[11].acc, "AccelVFD11",
		1.0, 1.0, 200.0,
		decFormat_None, k_factor, n_factor, valtypeUDINT, "VFD11(Forming Mesh CV) Acceleration [0.1 sec]");

	hmiParamListTableAddEntryNext(&gHmiParamTable,
		(UDINT)&pAppCfg->vfd[12].acc, "AccelVFD12",
		1.0, 1.0, 200.0,
		decFormat_None, k_factor, n_factor, valtypeUDINT, "VFD12(Exit Mesh CV) Acceleration [0.1 sec]");

	//Deceleration
	hmiParamListTableAddEntryNext(&gHmiParamTable,
		(UDINT)&pAppCfg->vfd[1].dec, "DecelVFD1",
		1.0, 0.0, 10.0,
		decFormat_None, k_factor, n_factor, valtypeUDINT, "VFD1(Elevator) Deceleration [0.1 sec]");

	hmiParamListTableAddEntryNext(&gHmiParamTable,
		(UDINT)&pAppCfg->vfd[2].dec, "DecelVFD2",
		1.0, 0.0, 20.0,
		decFormat_None, k_factor, n_factor, valtypeUDINT, "VFD2(Table) Deceleration [0.1 sec]");

	hmiParamListTableAddEntryNext(&gHmiParamTable,
		(UDINT)&pAppCfg->vfd[5].dec, "DecelVFD5",
		1.0, 0.0, 20.0,
		decFormat_None, k_factor, n_factor, valtypeUDINT, "VFD5(Row Forming Rollers) Deceleration [0.1 sec]");

	hmiParamListTableAddEntryNext(&gHmiParamTable,
		(UDINT)&pAppCfg->vfd[6].dec, "DecelVFD52",
		1.0, 0.0, 20.0,
		decFormat_None, k_factor, n_factor, valtypeUDINT, "VFD52(Row Forming Rollers 2) Deceleration [0.1 sec]");

	hmiParamListTableAddEntryNext(&gHmiParamTable,
		(UDINT)&pAppCfg->vfd[11].dec, "DecelVFD11",
		1.0, 0.0, 200.0,
		decFormat_None, k_factor, n_factor, valtypeUDINT, "VFD11(Forming Mesh CV) Deceleration [0.1 sec]");

	hmiParamListTableAddEntryNext(&gHmiParamTable,
		(UDINT)&pAppCfg->vfd[12].dec, "DecelVFD12",
		1.0, 0.0, 200.0,
		decFormat_None, k_factor, n_factor, valtypeUDINT, "VFD12(Exit Mesh CV) Deceleration [0.1 sec]");

	hmiParamListTableEntryLast(&gHmiParamTable);

}

static void hmiTableMachCfg()
{
	configApp_typ* pAppCfg = &gConfigApp;

	DINT decFormat_None = -2; //no dec places
	DINT decFormat_0 = -1;    //1 dec place
	//DINT decFormat_00 = 0;    //default (2) dec places as set in the control
//	DINT decFormat_000 = 1;    //3 dec places

	//scaling
	//y=kx+n where: y=HMI value, x=PLC value
	REAL k_factor = 1.0;
	REAL n_factor = 0.0;
	UINT valtypeUDINT = 0;//UDINT
	UINT valtypeREAL = 1;//REAL

	hmiParamListTableEntryFirst(&gHmiParamTable, "Mechanical Properties");

	hmiParamListTableAddEntryNext(&gHmiParamTable,
		(UDINT)&pAppCfg->options.optTearSheetEquiped, "TierSheetPresent",
		0.0, 0.0, 1.0,
		decFormat_None, k_factor, n_factor, valtypeUDINT, "1-Machine is equiped with a tier sheet inserting assembly.");

	hmiParamListTableAddEntryNext(&gHmiParamTable,
		(UDINT)&pAppCfg->options.optOption1Equiped, "Option1Present",
		0.0, 0.0, 1.0,
		decFormat_None, k_factor, n_factor, valtypeUDINT, "1-Machine is equipped with Option1 assembly.");

	hmiParamListTableAddEntryNext(&gHmiParamTable,
		(UDINT)&pAppCfg->options.palletDispenserOption, "PalletDispenserOption",
		0.0, 0.0, 1.0,
		decFormat_None, k_factor, n_factor, valtypeUDINT, "0-Pallet Dispenser Is NOT Present/NOT Equipped; 1-Pallet Dispenser is present/equipped.");

	hmiParamListTableAddEntryNext(&gHmiParamTable,
		(UDINT)&pAppCfg->options.frontSquaringOption, "FrontSquaringOption",
		0.0, 0.0, 1.0,
		decFormat_None, k_factor, n_factor, valtypeUDINT, "0-Front Squaring assembly Is NOT Present/NOT Equipped; 1-Front Squaring assembly is present/equipped.");

	hmiParamListTableAddEntryNext(&gHmiParamTable,
		(UDINT)&pAppCfg->system.boxInfeedSide, "InfeedLeftOrRight",
		0.0, 0.0, 1.0,
		decFormat_None, k_factor, n_factor, valtypeUDINT, "0-Box infeed Right to Left. 1-Box infeed Left to Right. Point of reference: person standing in front of the row pusher assembly looking towards the layer forming table.");

	hmiParamListTableAddEntryNext(&gHmiParamTable,
		(UDINT)&pAppCfg->system.simulationMode , "SimulationMode",
		0.0, 0.0, 1.0,
		decFormat_None, k_factor, n_factor, valtypeUDINT, "Simulation Mode. 0-OFF, 1-ON (Testing only!)");

	hmiParamListTableAddEntryNext(&gHmiParamTable,
		(UDINT)&pAppCfg->system.bladeStopCount, "NumberOfBladeStops",
		0.0, 0.0, 6.0,
		decFormat_None, k_factor, n_factor, valtypeUDINT, "Total number of blade stops on the machine.");

	hmiParamListTableAddEntryNext(&gHmiParamTable,
		(UDINT)&pAppCfg->system.bladeStopDistance[0] , "BladeStop1Distance",
		10.0, 0.0, 100.0,
		decFormat_0, k_factor, n_factor, valtypeREAL, "Distance/position of the blade stop 1 [inch]. Blade 1 is ALWAYS the blade closest to the infeed/incoming side of the row forming CV.");

	hmiParamListTableAddEntryNext(&gHmiParamTable,
		(UDINT)&pAppCfg->system.bladeStopDistance[1] , "BladeStop2Distance",
		12.0, 0.0, 100.0,
		decFormat_0, k_factor, n_factor, valtypeREAL, "Distance/position of the blade stop 2 [inch]");

	hmiParamListTableAddEntryNext(&gHmiParamTable,
		(UDINT)&pAppCfg->system.bladeStopDistance[2] , "BladeStop3Distance",
		14.0, 0.0, 100.0,
		decFormat_0, k_factor, n_factor, valtypeREAL, "Distance/position of the blade stop 3 [inch]");

	hmiParamListTableAddEntryNext(&gHmiParamTable,
		(UDINT)&pAppCfg->system.bladeStopDistance[3] , "BladeStop4Distance",
		16.0, 0.0, 100.0,
		decFormat_0, k_factor, n_factor, valtypeREAL, "Distance/position of the blade stop 4 [inch]");

	hmiParamListTableAddEntryNext(&gHmiParamTable,
		(UDINT)&pAppCfg->system.bladeStopDistance[4] , "BladeStop5Distance",
		18.0, 0.0, 100.0,
		decFormat_0, k_factor, n_factor, valtypeREAL, "Distance/position of the blade stop 5 [inch]");

	hmiParamListTableEntryLast(&gHmiParamTable);
}

//control visibility of the INPUT field (layer) for the parametar edit/view table
static void loginLevelParameterEditControl(UDINT minRights, UDINT minLevel)
{
	//controlling the locking of the editing form
	//(i.e. to lock > visibility set to 0 (visible) as the flag is used for a touch area over the inputs
	gHmiParamTable.selValueFormVisible = ((gPaiUserMgr.currentGroup.AccessRights[0] >= minRights) && (gPaiUserMgr.currentGroup.Level >= minLevel)) ? 1 : 0;
}

/*
###############################################################################
HMI screen handling logic
###############################################################################
*/
void screenHandlers(paiHmiTemplate_typ* pHmi)
{
	//Page specific init logic
	if(pHmi->prv.pageInit){
		//control visibility of the parametar input form

		//screen init event
		//define screen name
		switch(pHmi->runtime.pageCurrent){
			case SID_Settings_Timers:
			break;
			case SID_Settings_MachCfg:
				loginLevelParameterEditControl(mpUSER_ACCESS_FULL, 100); //only manufacturer
				hmiTableMachCfg();
			break;
			case SID_Settings_Options:
				loginLevelParameterEditControl(mpUSER_ACCESS_FULL, 100); //only manufacturer
				hmiTableOptions();
				break;
			case SID_Settings_VFDs:
				break;
			case SID_Recipe_PalletTimers:
				loginLevelParameterEditControl(mpUSER_ACCESS_FULL, 20); //normaly, supervisor is allowed to change data
				hmiTableRecipeTimers();
				break;
			case SID_Recipe_PalletVFDs:
				loginLevelParameterEditControl(mpUSER_ACCESS_FULL, 20); //normaly, supervisor is allowed to change data
				hmiTableRecipeVFDs();
				break;
			case SID_Main_Monitor:
			case SID_Recipe_PalletSelect:
			case SID_Recipe_PalletConfig:
			case SID_System_Files:
			case SID_Recipe_LayerDesign:
			case SID_Recipe_LayerPreview:
			case SID_Settings_System:
				loginLevelParameterEditControl(mpUSER_ACCESS_FULL, 10); //normaly, supervisor is allowed to change data
				break;
			case SID_Manual:
			case SID_Manual2:
				loginLevelParameterEditControl(mpUSER_ACCESS_FULL, 10); //normaly, supervisor is allowed to change data
				break;
			default:
			break;
		}
	}

	//Page specific cyclic logic
//	switch(page){
//		case SID_Workers_51:
//			screen_Workers_51();
//		break;
//		case SID_Setup_61:
//			screen_Setup_61();
//			break;
//	}

	hmiParamListTableCyclic(&gHmiParamTable);
}

/*
###############################################################################
HMI Logic: Running msg support (see screen saver)
###############################################################################
*/
void paiRunningMsgInit(paiHmiMsgRunning_typ* p, char* pMsg)
{
	if(!p)
		return;

	p->iMsgAddr = (UDINT)pMsg;
	p->curIdx = 0;
	p->state = 0;
}

void paiRunningMsgCyclic(paiHmiMsgRunning_typ* p)
{
	int lenMsg;
	int lenMax;
	int msgStartIdx;
	int msgCopyLen;

	if(!p || !p->iMsgAddr)
		return;

	bgTimerCyclic(&p->tmr1);

	if(!p->iEnable){
		p->oMsgVisible = 1;//not visible
		return;
	}
	p->oMsgVisible = 0;//visible

	if(!bgTimerIsTimeOut(&p->tmr1) ){
		return;
	}
	bgTimerStart(&p->tmr1, p->iScrollDelayXms);

	if(!p->state){
		p->curIdx++;
		if(p->curIdx >= p->iScrollLength){
			p->state = 1;
		}
	}else{
		p->curIdx--;
		if(p->curIdx == 0){
			p->state = 0;
		}
	}

	lenMax = paiHMI_ENUM_RUNMSG_MAXLEN - 1;
	lenMsg = brsstrlen((UDINT)p->iMsgAddr);
	msgStartIdx = (p->curIdx < lenMax) ? p->curIdx : lenMax;

	brsmemset((UDINT)p->oMsg, ' ', lenMax);
	p->oMsg[lenMax] = 0;

	msgCopyLen = 0;
	if(msgStartIdx < lenMax){
		msgCopyLen = (lenMax - msgStartIdx) < lenMsg ? (lenMax - msgStartIdx) : lenMsg;
	}
	brsmemcpy((UDINT)&p->oMsg[msgStartIdx], (UDINT)p->iMsgAddr, msgCopyLen);
}

/*
###############################################################################
HMI Logic: Layer editor HMI support
###############################################################################
*/
void appHmiLayerEditorCmdTxtGenCell(int row, int col)
{
	char txt[64];
	int 	cmdIdxBlade = gLayerEditor.palCfgRows[row].palCfgCmds[col].cmdBlade;
	int 	cmdIdxCase = gLayerEditor.palCfgRows[row].palCfgCmds[col].cmdCase;

	switch(cmdIdxCase){
		case 0:
			brsstrcpy((UDINT)txt, (UDINT)"");
			goto exitHere;
		break;
		case 1:
			brsstrcpy((UDINT)txt, (UDINT)"Case");
		break;
		case 2:
			brsstrcpy((UDINT)txt, (UDINT)"Case+90");
			break;
		case 3:
			brsstrcpy((UDINT)txt, (UDINT)"Case-90");
			break;
		case 4:
			brsstrcpy((UDINT)txt, (UDINT)"Case180");
			break;
		default:
			brsstrcpy((UDINT)txt, (UDINT)"Case???");
			break;
	}

	switch(cmdIdxBlade){
		case 0:
			break;
		case 1:
			brsstrcat((UDINT)txt, (UDINT)"\nBlade1");
			break;
		case 2:
			brsstrcat((UDINT)txt, (UDINT)"\nBlade2");
			break;
		case 3:
			brsstrcat((UDINT)txt, (UDINT)"\nBlade3");
			break;
		case 4:
			brsstrcat((UDINT)txt, (UDINT)"\nBlade4");
			break;
		case 5:
			brsstrcat((UDINT)txt, (UDINT)"\nBlade5");
			break;
		case 6:
			brsstrcat((UDINT)txt, (UDINT)"\nBlade6");
			break;
		default:
			brsstrcat((UDINT)txt, (UDINT)"\nBlade??");
			break;
	}

exitHere:
	brsstrcpy( (UDINT)gLayerEditorTxt.palCfgRowsTxt[row].palCfgCmdsTxt[col].cmdTxt, (UDINT)txt);
}

void appHmiLayerEditorCmdTxtGen()
{
	int ii;
	int row;
	int col;

	for(ii=0; ii<64; ii++){
		row = ii / 8;
		col = ii % 8;
		appHmiLayerEditorCmdTxtGenCell(row, col);
	}
}

void appHmiLayerEditorActiveCellBackClr()
{
	int ii;
	int row;
	int col;

	if(gLayerEditorTxt.curIdxEditorCell == gLayerEditorTxt.curIdxEditorCellOld)
		return;
	gLayerEditorTxt.curIdxEditorCellOld = gLayerEditorTxt.curIdxEditorCell;

	for(ii=0; ii<64; ii++){
		row = ii / 8;
		col = ii % 8;

		if(ii != gLayerEditorTxt.curIdxEditorCell){
			gLayerEditorTxt.palCfgRowsTxt[row].palCfgCmdsTxt[col].colorIdx = 0;
		}else{
			gLayerEditorTxt.palCfgRowsTxt[row].palCfgCmdsTxt[col].colorIdx = 1;
			gLayerEditorTxt.curIdxRow = row;
			gLayerEditorTxt.curIdxCmd = col;

			gLayerEditorTxt.cmdIdxBlade = gLayerEditor.palCfgRows[row].palCfgCmds[col].cmdBlade;
			gLayerEditorTxt.cmdIdxCase = gLayerEditor.palCfgRows[row].palCfgCmds[col].cmdCase;
			brsstrcpy((UDINT)gLayerEditorTxt.curCmdTxt, (UDINT)gLayerEditorTxt.palCfgRowsTxt[row].palCfgCmdsTxt[col].cmdTxt);
		}
	}
}

void appHmiLayerEditor()
{

	appHmiLayerEditorActiveCellBackClr();

	if(gLayerEditorTxt.cmdEntryCompletion){
		gLayerEditorTxt.cmdEntryCompletion = 0;
		gLayerEditor.palCfgRows[gLayerEditorTxt.curIdxRow].palCfgCmds[gLayerEditorTxt.curIdxCmd].cmdBlade = gLayerEditorTxt.cmdIdxBlade;
		gLayerEditor.palCfgRows[gLayerEditorTxt.curIdxRow].palCfgCmds[gLayerEditorTxt.curIdxCmd].cmdCase = gLayerEditorTxt.cmdIdxCase;
	}
	appHmiLayerEditorCmdTxtGenCell(gLayerEditorTxt.curIdxRow, gLayerEditorTxt.curIdxCmd);
	brsstrcpy((UDINT)gLayerEditorTxt.curCmdTxt, (UDINT)gLayerEditorTxt.palCfgRowsTxt[gLayerEditorTxt.curIdxRow].palCfgCmdsTxt[gLayerEditorTxt.curIdxCmd].cmdTxt);
}

/*
###############################################################################
HMI Logic: Layer Editor PV (gLayerEdit) Load/Save from/to a file
###############################################################################
*/
static void appHmiLayerFileHandlerLoadFilename(UDINT pFilename)
{
	int IDX_SERDES_ITEM = 2;

	brsstrcpy((UDINT)gPVSerDesMgr.pvItems[IDX_SERDES_ITEM].iFilename, (UDINT)pFilename);
	gPVSerDesMgr.pvItems[IDX_SERDES_ITEM].iDesRequest = 1;
	gPVSerDesMgr.pvItems[IDX_SERDES_ITEM].oDesCountOld = gPVSerDesMgr.pvItems[IDX_SERDES_ITEM].oDesCount;
}

static void appHmiLayerFileHandlerLoadCurSel()
{
int curSel;
int IDX_SERDES_ITEM = 2;

	curSel = gPaiMp.data.MpRecipeUIConnectCustom1.Recipe.List.SelectedIndex;
	if(curSel > gPaiMp.data.MpRecipeUIConnectCustom1.Recipe.List.MaxSelection){
		// Show the alert with a specified text and for a selected amount of time
		paiHmiAlertShow(&gPaiHmiAlertMsg, "WARNING:","Filename not selected!\nPlease select a filename from the list.", 3000);
		return;
	}
	if(gPaiMp.data.MpRecipeUIConnectCustom1.Recipe.List.Names[curSel][0] == 0){
		// Show the alert with a specified text and for a selected amount of time
		paiHmiAlertShow(&gPaiHmiAlertMsg, "WARNING:","Filename not defined!\nPlease select a filename from the list.", 3000);
		return;
	}
	brsstrcpy((UDINT)gPVSerDesMgr.pvItems[IDX_SERDES_ITEM].iFilename, (UDINT)gPaiMp.data.MpRecipeUIConnectCustom1.Recipe.List.Names[curSel]);
	gPVSerDesMgr.pvItems[IDX_SERDES_ITEM].iDesRequest = 1;
	gPVSerDesMgr.pvItems[IDX_SERDES_ITEM].oDesCountOld = gPVSerDesMgr.pvItems[IDX_SERDES_ITEM].oDesCount;
}

static void appHmiLayerFileHandlerCreateNew()
{
	int IDX_SERDES_ITEM = 2;

	if(gPaiMp.data.MpRecipeUIConnectCustom1.New.FileName[0] == 0){
		// Show the alert with a specified text and for a selected amount of time
		paiHmiAlertShow(&gPaiHmiAlertMsg, "WARNING:","New layer file not defined!\nPlease enter a file name.", 3000);
		return;
	}
	brsstrcpy((UDINT)gPVSerDesMgr.pvItems[IDX_SERDES_ITEM].iFilename, (UDINT)gPaiMp.data.MpRecipeUIConnectCustom1.New.FileName);
	brsstrcpy((UDINT)gLayerEditor.layerFilename, (UDINT)gPaiMp.data.MpRecipeUIConnectCustom1.New.FileName);
	gPVSerDesMgr.pvItems[IDX_SERDES_ITEM].iSerRequest = 1;
	gPVSerDesMgr.pvItems[IDX_SERDES_ITEM].oSerCountOld = gPVSerDesMgr.pvItems[IDX_SERDES_ITEM].oSerCount;
}

static void appHmiLayerFileHandlerSaveCurrent()
{
	int IDX_SERDES_ITEM = 2;

	if(gLayerEditor.layerFilename[0] == 0){
		// Show the alert with a specified text and for a selected amount of time
		paiHmiAlertShow(&gPaiHmiAlertMsg, "WARNING:","Filename not defined!\nPlease use Create to save these changes.", 3000);
		return;
	}
	brsstrcpy((UDINT)gPVSerDesMgr.pvItems[IDX_SERDES_ITEM].iFilename, (UDINT)gLayerEditor.layerFilename);
	gPVSerDesMgr.pvItems[IDX_SERDES_ITEM].iSerRequest = 1;
	gPVSerDesMgr.pvItems[IDX_SERDES_ITEM].oSerCountOld = gPVSerDesMgr.pvItems[IDX_SERDES_ITEM].oSerCount;
}

static void appHmiLayerFileHandlerCyclic()
{
	char txtMsg[255];
	int IDX_SERDES_ITEM = 2;

	if(gLayerFileHandler.iBtnLoad){
		gLayerFileHandler.iBtnLoad = 0;

		gLayerEditorTxt.curIdxEditorCell = 1000;
		gLayerEditorTxt.curIdxEditorCellOld = 0;

		appHmiLayerFileHandlerLoadCurSel();
	}

	if(gLayerFileHandler.iBtnLoadL1Preview){
		gLayerFileHandler.iBtnLoadL1Preview = 0;

		gLayerEditorTxt.curIdxEditorCell = 1000;
		gLayerEditorTxt.curIdxEditorCellOld = 0;

		appHmiLayerFileHandlerLoadFilename((UDINT)gPallete.palCfg.palLayerSettings[0].layerFilename);

		gPaiHmiMain.runtime.pageChange = 41;//layer preview page
	}

	if(gLayerFileHandler.iBtnLoadL2Preview){
		gLayerFileHandler.iBtnLoadL2Preview = 0;

		gLayerEditorTxt.curIdxEditorCell = 1000;
		gLayerEditorTxt.curIdxEditorCellOld = 0;

		appHmiLayerFileHandlerLoadFilename((UDINT)gPallete.palCfg.palLayerSettings[1].layerFilename);

		gPaiHmiMain.runtime.pageChange = 41;//layer preview page
	}

	if(gLayerFileHandler.iBtnNew){
		gLayerFileHandler.iBtnNew = 0;
		appHmiLayerFileHandlerCreateNew();
	}

	if(gLayerFileHandler.iBtnSave){
		gLayerFileHandler.iBtnSave = 0;
		appHmiLayerFileHandlerSaveCurrent();
	}

	//===================================
	//Check for file load/save events
	//===================================
	//check if PV restored from a file
	if(gPVSerDesMgr.pvItems[IDX_SERDES_ITEM].oDesCountOld != gPVSerDesMgr.pvItems[IDX_SERDES_ITEM].oDesCount){
		gPVSerDesMgr.pvItems[IDX_SERDES_ITEM].oDesCountOld = gPVSerDesMgr.pvItems[IDX_SERDES_ITEM].oDesCount;

		gLayerEditorTxt.curIdxEditorCell = 0;
		gLayerEditorTxt.curIdxEditorCellOld = 1000;

		//rebuild current layer editor view
		appHmiLayerEditorCmdTxtGen();
		brsstrcpy((UDINT)txtMsg, "Layer program loaded from a file!\n\nFilename: ");
		brsstrcat((UDINT)txtMsg, (UDINT)gPVSerDesMgr.pvItems[IDX_SERDES_ITEM].iFilename);
		paiHmiAlertShow(&gPaiHmiAlertMsg, "MESSAGE:", txtMsg, 3000);
		brsstrcpy((UDINT)gLayerEditor.layerFilename, (UDINT)gPVSerDesMgr.pvItems[2].iFilename);

		//trigger canvas redraw of the layer
		gCtrl.main.gCamApp_btnPreview = 1;
	}

	if(gPVSerDesMgr.pvItems[IDX_SERDES_ITEM].oSerCountOld != gPVSerDesMgr.pvItems[IDX_SERDES_ITEM].oSerCount){
		gPVSerDesMgr.pvItems[IDX_SERDES_ITEM].oSerCountOld = gPVSerDesMgr.pvItems[IDX_SERDES_ITEM].oSerCount;
		//rebuild current layer editor view
		appHmiLayerEditorCmdTxtGen();
		brsstrcpy((UDINT)txtMsg, "Layer program saved to a file!\n\nFilename: ");
		brsstrcat((UDINT)txtMsg, (UDINT)gPVSerDesMgr.pvItems[IDX_SERDES_ITEM].iFilename);
		paiHmiAlertShow(&gPaiHmiAlertMsg, "MESSAGE:", txtMsg, 3000);
		brsstrcpy((UDINT)gLayerEditor.layerFilename, (UDINT)gPVSerDesMgr.pvItems[IDX_SERDES_ITEM].iFilename);
		//refresh file viewer
		gPaiMp.data.MpRecipeUIConnectCustom1.Recipe.Refresh = 1;
	}

}

/*
###############################################################################
HMI Logic: Pallete recipe utility functions.
###############################################################################
*/
static void appHmiInitPalleteCfg()
{
	int ii;

	gPallete.palCfg.palLayerSettings[0].sameAsOtherLayer = 0;
	gPallete.palCfg.palLayerSettings[0].sameAsOtherLayer = 0;
	for(ii=2; ii<gPallete.palCfg.palActiveLayers; ii++){
		gPallete.palCfg.palLayerSettings[ii].sameAsOtherLayer = 1;
	}
}

static void appHmiSetPalleteLayersCfgL0Only()
{
	int ii;

	for(ii=1; ii<gPallete.palCfg.palActiveLayers; ii++){
		gPallete.palCfg.palLayerSettings[ii].sameAsOtherLayer = 1;
		gPallete.palCfg.palLayerSettings[ii].otherLayerIdx = 0;
	}
}

static BOOL appHmiIsLayerL1ProgramRequired()
{
	if(gPallete.palCfg.palLayerSettings[1].layerFilename[0] != 0)
		return 1;

	return 0;
}

static BOOL appHmiIsLayerL1RefExist()
{
int ii;

	for(ii=2; ii<gPallete.palCfg.palActiveLayers; ii++){
		if(gPallete.palCfg.palLayerSettings[ii].otherLayerIdx != 0)
			return 1;
	}
	return 0;
}

/*
###############################################################################
HMI Logic: Support from loadig Layer configuration PV-s (gLayer1 and gLayer2)
based on the information contained within a pallete recipe
###############################################################################
*/

static void appHmiLayerL0L1LoadRequest()
{
	gLayer_L0_L1_FileHandler.iBtnLoad = 1;
}

static BOOL appHmiLayerL0L1IsLoadRequested()
{
	if(gLayer_L0_L1_FileHandler.iBtnLoad){
		gLayer_L0_L1_FileHandler.iBtnLoad = 0;
		return 1;
	}
	return 0;
}

static void	appHmiSetLayerPrograms()
{

int ii;

	//layer[0] = always from file layerLO
	brsmemcpy( (UDINT)&gPallete.palCfgLayers[0], (UDINT)&gLayer_L0, sizeof(gLayer_L0));

	//layer 1 - if sameAsOtherLayer > it must be from layerLO file
	if(gPallete.palCfg.palLayerSettings[1].sameAsOtherLayer){
		brsmemcpy( (UDINT)&gPallete.palCfgLayers[1], (UDINT)&gLayer_L0, sizeof(gLayer_L0));
	}else{
		brsmemcpy( (UDINT)&gPallete.palCfgLayers[1], (UDINT)&gLayer_L1, sizeof(gLayer_L1));
	}

	//other active layers; check what layer used, copy required layer data
	for(ii=2; ii < gPallete.palCfg.palActiveLayers; ii++){
		if(gPallete.palCfg.palLayerSettings[ii].otherLayerIdx){
			brsmemcpy( (UDINT)&gPallete.palCfgLayers[ii], (UDINT)&gLayer_L1, sizeof(gLayer_L1));
		}else{
			brsmemcpy( (UDINT)&gPallete.palCfgLayers[ii], (UDINT)&gLayer_L0, sizeof(gLayer_L0));
		}
	}

	for(ii=gPallete.palCfg.palActiveLayers; ii < APP_REC_MAXLAYER; ii++){
			brsmemset( (UDINT)&gPallete.palCfgLayers[ii], 0, sizeof(gLayer_L0));
	}

}

static void appHmiLayerL0L1FileLoadingCyclic()
{
int curSel;
char txtMsg[255];
int IDX_SERDES_ITEM = 4;

	bgTimerCyclic(&gLayer_L0_L1_FileHandler.fileHandlerTimer);

	switch(gLayer_L0_L1_FileHandler.fileHandlerState){
		case 0:
			if( !appHmiLayerL0L1IsLoadRequested() )
				return;

			appHmiInitPalleteCfg();

			gLayer_L0_L1_FileHandler.fileHandlerState = 10;
			bgTimerStart(&gLayer_L0_L1_FileHandler.fileHandlerTimer, 2500);

		break;
		case 10:
			if(!bgTimerIsTimeOut(&gLayer_L0_L1_FileHandler.fileHandlerTimer))
				return;

			//try to load L0 layer configuration
			if(gPallete.palCfg.palLayerSettings[0].layerFilename[0] == 0){
				// Show the alert with a specified text and for a selected amount of time
				paiHmiAlertShow(&gPaiHmiAlertMsg, "ERROR:","Layer L0 filename is not defined!\nInvalid pallete recipe file.", 3000);
				gPallete.ctrlProc.oPalleteRecipeIsValid = 0;
				gLayer_L0_L1_FileHandler.fileHandlerState = 50;
				return;
			}
			IDX_SERDES_ITEM = 4;
			brsstrcpy((UDINT)gPVSerDesMgr.pvItems[IDX_SERDES_ITEM].iFilename, (UDINT)gPallete.palCfg.palLayerSettings[0].layerFilename);
			gPVSerDesMgr.pvItems[IDX_SERDES_ITEM].iDesRequest = 1;
			gPVSerDesMgr.pvItems[IDX_SERDES_ITEM].oDesCountOld = gPVSerDesMgr.pvItems[IDX_SERDES_ITEM].oDesCount;
			gPVSerDesMgr.pvItems[IDX_SERDES_ITEM].oErrorCountOld = gPVSerDesMgr.pvItems[IDX_SERDES_ITEM].oErrorCount;
			gLayer_L0_L1_FileHandler.fileHandlerState = 20;
		break;
		case 20:
			IDX_SERDES_ITEM = 4;
			if(gPVSerDesMgr.pvItems[IDX_SERDES_ITEM].oDesCountOld != gPVSerDesMgr.pvItems[IDX_SERDES_ITEM].oDesCount){
				brsstrcpy((UDINT)txtMsg, "Layer L0 program loaded from a file!\n\nFilename: ");
				brsstrcat((UDINT)txtMsg, (UDINT)gPVSerDesMgr.pvItems[IDX_SERDES_ITEM].iFilename);
				paiHmiAlertShow(&gPaiHmiAlertMsg, "MESSAGE:", txtMsg, 2000);
				bgTimerStart(&gLayer_L0_L1_FileHandler.fileHandlerTimer, 2500);
				gLayer_L0_L1_FileHandler.fileHandlerState = 30;
			}

			if(gPVSerDesMgr.pvItems[IDX_SERDES_ITEM].oErrorCountOld != gPVSerDesMgr.pvItems[IDX_SERDES_ITEM].oErrorCount){
				paiHmiAlertShow(&gPaiHmiAlertMsg, "ERROR:","Layer L0 program load error!\nPallete recipe is NOT valid.\nPlease use a different pallete recipe.", 3000);
				gPallete.ctrlProc.oPalleteRecipeIsValid = 0;
				gLayer_L0_L1_FileHandler.fileHandlerState = 50;
			}
			break;
		case 30:
			if(!bgTimerIsTimeOut(&gLayer_L0_L1_FileHandler.fileHandlerTimer))
				return;

			if(!appHmiIsLayerL1ProgramRequired() && !appHmiIsLayerL1RefExist()){
				// Show the alert with a specified text and for a selected amount of time
				paiHmiAlertShow(&gPaiHmiAlertMsg, "WARNING:","Layer L1 is NOT used!\n", 3000);
				gLayer_L0_L1_FileHandler.fileHandlerState = 50;
				return;
			}
			if(!appHmiIsLayerL1ProgramRequired() && appHmiIsLayerL1RefExist()){
				// Show the alert with a specified text and for a selected amount of time
				paiHmiAlertShow(&gPaiHmiAlertMsg, "ERROR:","Layer L1 referenced but not defined!\nInvalid pallete recipe file.", 3000);
				gPallete.ctrlProc.oPalleteRecipeIsValid = 0;
				gLayer_L0_L1_FileHandler.fileHandlerState = 50;
				return;
			}
			IDX_SERDES_ITEM = 5;
			brsstrcpy((UDINT)gPVSerDesMgr.pvItems[IDX_SERDES_ITEM].iFilename, (UDINT)gPallete.palCfg.palLayerSettings[1].layerFilename);
			gPVSerDesMgr.pvItems[IDX_SERDES_ITEM].iDesRequest = 1;
			gPVSerDesMgr.pvItems[IDX_SERDES_ITEM].oDesCountOld = gPVSerDesMgr.pvItems[IDX_SERDES_ITEM].oDesCount;
			gPVSerDesMgr.pvItems[IDX_SERDES_ITEM].oErrorCountOld = gPVSerDesMgr.pvItems[IDX_SERDES_ITEM].oErrorCount;
			gLayer_L0_L1_FileHandler.fileHandlerState = 40;

			break;
		case 40:
			IDX_SERDES_ITEM = 5;
			if(gPVSerDesMgr.pvItems[IDX_SERDES_ITEM].oDesCountOld != gPVSerDesMgr.pvItems[IDX_SERDES_ITEM].oDesCount){
				brsstrcpy((UDINT)txtMsg, "Layer L1 program loaded from a file!\n\nFilename: ");
				brsstrcat((UDINT)txtMsg, (UDINT)gPVSerDesMgr.pvItems[IDX_SERDES_ITEM].iFilename);
				paiHmiAlertShow(&gPaiHmiAlertMsg, "MESSAGE:", txtMsg, 2000);
				bgTimerStart(&gLayer_L0_L1_FileHandler.fileHandlerTimer, 2500);
				gLayer_L0_L1_FileHandler.fileHandlerState = 50;
			}

			if(gPVSerDesMgr.pvItems[IDX_SERDES_ITEM].oErrorCountOld != gPVSerDesMgr.pvItems[IDX_SERDES_ITEM].oErrorCount){
				paiHmiAlertShow(&gPaiHmiAlertMsg, "ERROR:","Layer L1 program load error!\nPallete recipe is NOT valid.\nPlease use a different pallete recipe.", 3000);
				gPallete.ctrlProc.oPalleteRecipeIsValid = 0;
				gLayer_L0_L1_FileHandler.fileHandlerState = 50;
			}
			break;
			break;
		case 50:
			bgTimerStart(&gLayer_L0_L1_FileHandler.fileHandlerTimer, 2500);
			gLayer_L0_L1_FileHandler.fileHandlerState = 51;
			break;
		case 51:
			if(!bgTimerIsTimeOut(&gLayer_L0_L1_FileHandler.fileHandlerTimer))
				return;

			if(gPallete.ctrlProc.oPalleteRecipeIsValid){
				//paiHmiAlertShow(&gPaiHmiAlertMsg, "INFO:","Layer L1 program load error!\nPallete recipe is NOT valid.\nPlease use a different pallete recipe.", 1000);
				appHmiSetLayerPrograms();
			}else{
				paiHmiAlertShow(&gPaiHmiAlertMsg, "ERROR:","Loaded pallete recipe is not valid!\nPlease use/create a different pallete recipe.", 5000);
			}
			gLayer_L0_L1_FileHandler.fileHandlerState = 0;
			break;
	}
}
/*
###############################################################################
HMI Logic: Pallete configuration recipe PV (gPallete.palCfg) Load/Save from/to a file
###############################################################################
*/
static void appHmiPalleteFileHandlerLoadCurrent()
{
	int curSel;
	int IDX_SERDES_ITEM = 3;

	curSel = gPaiMp.data.MpRecipeUIConnectCustom2.Recipe.List.SelectedIndex;
	if(curSel > gPaiMp.data.MpRecipeUIConnectCustom2.Recipe.List.MaxSelection){
		// Show the alert with a specified text and for a selected amount of time
		paiHmiAlertShow(&gPaiHmiAlertMsg, "WARNING:","Filename not selected!\nPlease select a filename from the list.", 3000);
		return;
	}
	if(gPaiMp.data.MpRecipeUIConnectCustom2.Recipe.List.Names[curSel][0] == 0){
		// Show the alert with a specified text and for a selected amount of time
		paiHmiAlertShow(&gPaiHmiAlertMsg, "WARNING:","Filename not defined!\nPlease select a filename from the list.", 3000);
		return;
	}
	brsstrcpy((UDINT)gPVSerDesMgr.pvItems[IDX_SERDES_ITEM].iFilename, (UDINT)gPaiMp.data.MpRecipeUIConnectCustom2.Recipe.List.Names[curSel]);
	gPVSerDesMgr.pvItems[IDX_SERDES_ITEM].iDesRequest = 1;
	gPVSerDesMgr.pvItems[IDX_SERDES_ITEM].oDesCountOld = gPVSerDesMgr.pvItems[IDX_SERDES_ITEM].oDesCount;

	//gSerDesHMI_gPalletCfg.iBtnDesRequest = 1;

}

static void appHmiPalleteFileHandlerCreateNew()
{
	int curSel;
	int IDX_SERDES_ITEM = 3;

	if(gPaiMp.data.MpRecipeUIConnectCustom2.New.FileName[0] == 0){
		// Show the alert with a specified text and for a selected amount of time
		paiHmiAlertShow(&gPaiHmiAlertMsg, "WARNING:","New layer file not defined!\nPlease enter a file name.", 3000);
		return;
	}
	brsstrcpy((UDINT)gPVSerDesMgr.pvItems[IDX_SERDES_ITEM].iFilename, (UDINT)gPaiMp.data.MpRecipeUIConnectCustom2.New.FileName);
	brsstrcpy((UDINT)gPallete.palCfg.palFilename, (UDINT)gPaiMp.data.MpRecipeUIConnectCustom2.New.FileName);
	gPVSerDesMgr.pvItems[IDX_SERDES_ITEM].iSerRequest = 1;
	gPVSerDesMgr.pvItems[IDX_SERDES_ITEM].oSerCountOld = gPVSerDesMgr.pvItems[IDX_SERDES_ITEM].oSerCount;
	//gSerDesHMI_gPalletCfg.iBtnSerRequest = 1;

}

static void appHmiPalleteFileHandlerSaveCurrent()
{
	int IDX_SERDES_ITEM = 3;

	if(gPallete.palCfg.palFilename[0] == 0){
		// Show the alert with a specified text and for a selected amount of time
		paiHmiAlertShow(&gPaiHmiAlertMsg, "WARNING:","Filename not defined!\nPlease use Create to save changes.", 3000);
		return;
	}
	brsstrcpy((UDINT)gPVSerDesMgr.pvItems[IDX_SERDES_ITEM].iFilename, (UDINT)gPallete.palCfg.palFilename);
	gPVSerDesMgr.pvItems[IDX_SERDES_ITEM].iSerRequest = 1;
	gPVSerDesMgr.pvItems[IDX_SERDES_ITEM].oSerCountOld = gPVSerDesMgr.pvItems[IDX_SERDES_ITEM].oSerCount;
	//gSerDesHMI_gPalletCfg.iBtnSerRequest = 1;

}

static void appHmiPalleteFileHandlerCyclic()
{
	char txtMsg[255];
	int IDX_SERDES_ITEM = 3;

	if(gPalleteFileHandler.iBtnLoad){
		gPalleteFileHandler.iBtnLoad = 0;
		appHmiPalleteFileHandlerLoadCurrent();
	}

	if(gPalleteFileHandler.iBtnNew){
		gPalleteFileHandler.iBtnNew = 0;
		appHmiPalleteFileHandlerCreateNew();
	}

	if(gPalleteFileHandler.iBtnSave){
		gPalleteFileHandler.iBtnSave = 0;
		appHmiPalleteFileHandlerSaveCurrent();
	}

	//===================================
	//Check for patter file PV-s load/save events
	//===================================
	//check if PV restored from a file
	if(gPVSerDesMgr.pvItems[IDX_SERDES_ITEM].oDesCountOld != gPVSerDesMgr.pvItems[IDX_SERDES_ITEM].oDesCount){
		gPVSerDesMgr.pvItems[IDX_SERDES_ITEM].oDesCountOld = gPVSerDesMgr.pvItems[IDX_SERDES_ITEM].oDesCount;
		//rebuild current layer editor view
		appHmiLayerEditorCmdTxtGen();
		brsstrcpy((UDINT)txtMsg, "Pattern program loaded from a file!\n\nFilename: ");
		brsstrcat((UDINT)txtMsg, (UDINT)gPVSerDesMgr.pvItems[IDX_SERDES_ITEM].iFilename);
		paiHmiAlertShow(&gPaiHmiAlertMsg, "MESSAGE:", txtMsg, 2000);
		brsstrcpy((UDINT)gPallete.palCfg.palFilename, (UDINT)gPVSerDesMgr.pvItems[IDX_SERDES_ITEM].iFilename);
		//mark recipe as valid
		gPallete.ctrlProc.oPalleteRecipeIsValid = 1;
		//start layer program loading; during that process, the above valid flag may get reset to 0!
		appHmiLayerL0L1LoadRequest();
		//GB: magic write
		*((UDINT*)gPVSerDesMgr.pvItems[IDX_SERDES_ITEM].optInitAtPowerUp.pTestDataStorage) = gPVSerDesMgr.pvItems[IDX_SERDES_ITEM].optInitAtPowerUp.iTestData;
	}

	if(gPVSerDesMgr.pvItems[IDX_SERDES_ITEM].oSerCountOld != gPVSerDesMgr.pvItems[IDX_SERDES_ITEM].oSerCount){
		gPVSerDesMgr.pvItems[IDX_SERDES_ITEM].oSerCountOld = gPVSerDesMgr.pvItems[IDX_SERDES_ITEM].oSerCount;
		//rebuild current layer editor view
		appHmiLayerEditorCmdTxtGen();
		brsstrcpy((UDINT)txtMsg, (UDINT)"Patttern program saved to a file!\n\nFilename: ");
		brsstrcat((UDINT)txtMsg, (UDINT)gPVSerDesMgr.pvItems[IDX_SERDES_ITEM].iFilename);
		paiHmiAlertShow(&gPaiHmiAlertMsg, "MESSAGE:", txtMsg, 3000);
		//refresh file viewer
		gPaiMp.data.MpRecipeUIConnectCustom2.Recipe.Refresh = 1;
		//GB: magic write
		*((UDINT*)gPVSerDesMgr.pvItems[IDX_SERDES_ITEM].optInitAtPowerUp.pTestDataStorage) = gPVSerDesMgr.pvItems[IDX_SERDES_ITEM].optInitAtPowerUp.iTestData;
	}

}

/*
###############################################################################
HMI Logic: Pallete Editor
###############################################################################
*/
void appHmiPalleteEditorVisibility()
{
	int ii;

	//control visibility of the pallete editor components
	for(ii=0; ii < 12; ii++){//todo: use const here
		if(ii < gPallete.palCfg.palActiveLayers){
			//visible
			gPallete.ctrlLayers[ii].layerVisible = 0;
			if(gConfigApp.options.optTearSheetEquiped){
				gPallete.ctrlLayers[ii].tearSheetOptionVisible = 0;
			}else{
				gPallete.ctrlLayers[ii].tearSheetOptionVisible = 1;
			}
			if(gConfigApp.options.optOption1Equiped){
				gPallete.ctrlLayers[ii].option1Visible = 0;
			}else{
				gPallete.ctrlLayers[ii].option1Visible = 1;
			}
		}else{
			//not visible
			gPallete.ctrlLayers[ii].layerVisible = 1;
			gPallete.ctrlLayers[ii].tearSheetOptionVisible = 1;
			gPallete.ctrlLayers[ii].option1Visible = 1;
		}
	}
}

static void appHmiPalleteEditorAssignLayerProgram()
{
	int curSel;

	if(gPallete.ctrlLayers[0].btnAssignLayerFilename){
		gPallete.ctrlLayers[0].btnAssignLayerFilename = 0;
		curSel = gPaiMp.data.MpRecipeUIConnectCustom1.Recipe.List.SelectedIndex;
		if(curSel > gPaiMp.data.MpRecipeUIConnectCustom1.Recipe.List.MaxSelection){
			// Show the alert with a specified text and for a selected amount of time
			paiHmiAlertShow(&gPaiHmiAlertMsg, "WARNING:","Filename not selected!\nPlease select a filename from the list.", 3000);
			return;
		}
		if(gPaiMp.data.MpRecipeUIConnectCustom1.Recipe.List.Names[curSel][0] == 0){
			// Show the alert with a specified text and for a selected amount of time
			paiHmiAlertShow(&gPaiHmiAlertMsg, "WARNING:","Filename not defined!\nPlease select a filename from the list.", 3000);
			return;
		}
		brsstrcpy((UDINT)gPallete.palCfg.palLayerSettings[0].layerFilename, (UDINT)gPaiMp.data.MpRecipeUIConnectCustom1.Recipe.List.Names[curSel]);
	}

	if(gPallete.ctrlLayers[1].btnAssignLayerFilename){
		gPallete.ctrlLayers[1].btnAssignLayerFilename = 0;
		curSel = gPaiMp.data.MpRecipeUIConnectCustom1.Recipe.List.SelectedIndex;
		if(curSel > gPaiMp.data.MpRecipeUIConnectCustom1.Recipe.List.MaxSelection){
			// Show the alert with a specified text and for a selected amount of time
			paiHmiAlertShow(&gPaiHmiAlertMsg, "WARNING:","Filename not selected!\nPlease select a filename from the list.", 3000);
			return;
		}
		if(gPaiMp.data.MpRecipeUIConnectCustom1.Recipe.List.Names[curSel][0] == 0){
			// Show the alert with a specified text and for a selected amount of time
			paiHmiAlertShow(&gPaiHmiAlertMsg, "WARNING:","Filename not defined!\nPlease select a filename from the list.", 3000);
			return;
		}
		brsstrcpy((UDINT)gPallete.palCfg.palLayerSettings[1].layerFilename, (UDINT)gPaiMp.data.MpRecipeUIConnectCustom1.Recipe.List.Names[curSel]);
		gPallete.palCfg.palLayerSettings[1].sameAsOtherLayer = 0;
	}

	if(gPallete.ctrlLayers[1].btnDeleteLayerFilename){
		gPallete.ctrlLayers[1].btnDeleteLayerFilename = 0;

		if(gPallete.palCfg.palLayerSettings[1].layerFilename[0] != 0){
			paiHmiDialogShow(&gPaiHmiDialogMsg, "Delete layer L1 program filename and remove all reference to L1?", 10000, DLG_DeleteL1FilenameOK, DLG_DeleteL1FilenameCancel, 1);
		}
	}

	if(gPaiHmiDialogMsg.result == DLG_DeleteL1FilenameOK){
		gPaiHmiDialogMsg.result = 0;
		gPallete.palCfg.palLayerSettings[1].layerFilename[0] = 0;
		appHmiSetPalleteLayersCfgL0Only();
	}
	if(gPaiHmiDialogMsg.result == DLG_DeleteL1FilenameCancel){
		gPaiHmiDialogMsg.result = 0;
	}

}

void appHmiPalleteEditorCyclic()
{

	appHmiPalleteEditorVisibility();
	appHmiPalleteEditorAssignLayerProgram();

}

void appScalingAndConversion()
{
	gCtrl.retainerbar.barDwDlyTmXms = (UDINT)(gPallete.palCfg.palSettings.timers.onDlyPRRetBarDown * 1000.0);
}

void appBladeStopsUsed()
{
	switch(gConfigApp.system.bladeStopCount){
		case 0:
			gCtrl.rowforming.isStopBladeUsed1 = 0;
			gCtrl.rowforming.isStopBladeUsed2 = 0;
			gCtrl.rowforming.isStopBladeUsed3 = 0;
			gCtrl.rowforming.isStopBladeUsed4 = 0;
			gCtrl.rowforming.isStopBladeUsed5 = 0;
			gCtrl.rowforming.isStopBladeUsed6 = 0;
		break;
		case 1:
			gCtrl.rowforming.isStopBladeUsed1 = 1;
			gCtrl.rowforming.isStopBladeUsed2 = 0;
			gCtrl.rowforming.isStopBladeUsed3 = 0;
			gCtrl.rowforming.isStopBladeUsed4 = 0;
			gCtrl.rowforming.isStopBladeUsed5 = 0;
			gCtrl.rowforming.isStopBladeUsed6 = 0;
			break;
		case 2:
			gCtrl.rowforming.isStopBladeUsed1 = 1;
			gCtrl.rowforming.isStopBladeUsed2 = 1;
			gCtrl.rowforming.isStopBladeUsed3 = 0;
			gCtrl.rowforming.isStopBladeUsed4 = 0;
			gCtrl.rowforming.isStopBladeUsed5 = 0;
			gCtrl.rowforming.isStopBladeUsed6 = 0;
			break;
		case 3:
			gCtrl.rowforming.isStopBladeUsed1 = 1;
			gCtrl.rowforming.isStopBladeUsed2 = 1;
			gCtrl.rowforming.isStopBladeUsed3 = 1;
			gCtrl.rowforming.isStopBladeUsed4 = 0;
			gCtrl.rowforming.isStopBladeUsed5 = 0;
			gCtrl.rowforming.isStopBladeUsed6 = 0;
			break;
		case 4:
			gCtrl.rowforming.isStopBladeUsed1 = 1;
			gCtrl.rowforming.isStopBladeUsed2 = 1;
			gCtrl.rowforming.isStopBladeUsed3 = 1;
			gCtrl.rowforming.isStopBladeUsed4 = 1;
			gCtrl.rowforming.isStopBladeUsed5 = 0;
			gCtrl.rowforming.isStopBladeUsed6 = 0;
			break;
		case 5:
			gCtrl.rowforming.isStopBladeUsed1 = 1;
			gCtrl.rowforming.isStopBladeUsed2 = 1;
			gCtrl.rowforming.isStopBladeUsed3 = 1;
			gCtrl.rowforming.isStopBladeUsed4 = 1;
			gCtrl.rowforming.isStopBladeUsed5 = 1;
			gCtrl.rowforming.isStopBladeUsed6 = 0;
			break;
		case 6:
			gCtrl.rowforming.isStopBladeUsed1 = 1;
			gCtrl.rowforming.isStopBladeUsed2 = 1;
			gCtrl.rowforming.isStopBladeUsed3 = 1;
			gCtrl.rowforming.isStopBladeUsed4 = 1;
			gCtrl.rowforming.isStopBladeUsed5 = 1;
			gCtrl.rowforming.isStopBladeUsed6 = 1;
			break;
	}
}

void appVisibilityCaseInfeedSide()
{
	if(gConfigApp.system.boxInfeedSide == 0){
		gCtrl.main.visibleCaseInfeedOnLeft = 1;
		gCtrl.main.visibleCaseInfeedOnRight = 0;
	}else{
		gCtrl.main.visibleCaseInfeedOnLeft = 0;
		gCtrl.main.visibleCaseInfeedOnRight = 1;
	}
}

/*
###############################################################################
Logic to change to Alarm screen when alarm pops up
###############################################################################
*/
static void appHmiGotoAlarmScreen()
{
	static BOOL alarmIsTriggered;//remeber if switch to alarm page took place in order to allow going to other pages when alarm is active/present

	//switch to alarm screen when alarm pops up;
	if(!alarmIsTriggered && gAlarms.oIsAlarmActive && gAlarms.oIsAlarmNotAck && (gPaiHmiMain.runtime.pageCurrent != SID_Diag_Alarms) && (gPaiHmiMain.runtime.pageChange == -1)){
		gPaiHmiMain.runtime.pageChange = SID_Diag_Alarms;
		alarmIsTriggered = 1;
	}

	//reset alarm is triggered when no active alarms
	if(!gAlarms.oIsAlarmActive){
		alarmIsTriggered = 0;
	}

	//switch automatically back to main page when alarms are clear
	if(!alarmIsTriggered && !gAlarms.oIsAlarmActive && !gAlarms.oIsAlarmNotAck && (gPaiHmiMain.runtime.pageCurrent == SID_Diag_Alarms) && (gPaiHmiMain.runtime.pageChange == -1)){
		//9/21/2016; Following line commented out on the request from customer (David@ABC, based on the input from the end user (Duckhorn)
		//gPaiHmiMain.runtime.pageChange = SID_Main;

	}

}

/*
###############################################################################
Configuration file gConfig HMI logic
###############################################################################
*/
static void appHmiAppConfigFileLoadRequest()
{
	int IDX_SERDES_ITEM = 0;

	gPVSerDesMgr.pvItems[IDX_SERDES_ITEM].iDesRequest = 1;
	gPVSerDesMgr.pvItems[IDX_SERDES_ITEM].oDesCountOld = gPVSerDesMgr.pvItems[IDX_SERDES_ITEM].oDesCount;
}

static void appHmiAppConfigFileSaveRequest()
{
	int IDX_SERDES_ITEM = 0;

	gPVSerDesMgr.pvItems[IDX_SERDES_ITEM].optChangeMonitor.iChngAccepted = 1;
	gPVSerDesMgr.pvItems[IDX_SERDES_ITEM].oSerCountOld = gPVSerDesMgr.pvItems[IDX_SERDES_ITEM].oSerCount;
}

static void appHmiPalletRecipeFileSaveRequest()
{
	int IDX_SERDES_ITEM = 3;

	gPVSerDesMgr.pvItems[IDX_SERDES_ITEM].optChangeMonitor.iChngAccepted = 1;
	gPVSerDesMgr.pvItems[IDX_SERDES_ITEM].oSerCountOld = gPVSerDesMgr.pvItems[IDX_SERDES_ITEM].oSerCount;
}

static void appHmiAppConfigCancelChange()
{
	int IDX_SERDES_ITEM = 0;
	gPVSerDesMgr.pvItems[IDX_SERDES_ITEM].optChangeMonitor.iChngRejected = 1;
}

static void appHmiPalletRecipeCancelChange()
{
	int IDX_SERDES_ITEM = 3;
	gPVSerDesMgr.pvItems[IDX_SERDES_ITEM].optChangeMonitor.iChngRejected = 1;
}

static BOOL appHmiIsAppConfigChanged()
{
	int IDX_SERDES_ITEM = 0;
	return(gPVSerDesMgr.pvItems[IDX_SERDES_ITEM].optChangeMonitor.oChngDetected);
}

//check if PV restored from a file
static void appHmiAppConfigFileLoadEventCyclic()
{
	char txtMsg[255];
	int IDX_SERDES_ITEM = 0;

	if(gPVSerDesMgr.pvItems[IDX_SERDES_ITEM].oDesCountOld == gPVSerDesMgr.pvItems[IDX_SERDES_ITEM].oDesCount)
		return;

	gPVSerDesMgr.pvItems[IDX_SERDES_ITEM].oDesCountOld = gPVSerDesMgr.pvItems[IDX_SERDES_ITEM].oDesCount;
	brsstrcpy((UDINT)txtMsg, "Application configuration loaded from file.\n\nFilename: ");
	brsstrcat((UDINT)txtMsg, (UDINT)gPVSerDesMgr.pvItems[IDX_SERDES_ITEM].iFilename);
	paiHmiAlertShow(&gPaiHmiAlertMsg, "MESSAGE:", txtMsg, 3000);
}

static void appHmiAppConfigFileSaveEventCyclic()
{
	char txtMsg[255];
	int IDX_SERDES_ITEM = 0;

	if(gPVSerDesMgr.pvItems[IDX_SERDES_ITEM].oSerCountOld == gPVSerDesMgr.pvItems[IDX_SERDES_ITEM].oSerCount)
		return;

	gPVSerDesMgr.pvItems[IDX_SERDES_ITEM].oSerCountOld = gPVSerDesMgr.pvItems[IDX_SERDES_ITEM].oSerCount;
	brsstrcpy((UDINT)txtMsg, (UDINT)"Application configuration saved to file.\n\nFilename: ");
	brsstrcat((UDINT)txtMsg, (UDINT)gPVSerDesMgr.pvItems[IDX_SERDES_ITEM].iFilename);
	paiHmiAlertShow(&gPaiHmiAlertMsg, "MESSAGE:", txtMsg, 3000);
}

static void appHmiPalletRecipeFileSaveEventCyclic()
{
	char txtMsg[255];
	int IDX_SERDES_ITEM = 3;

	if(gPVSerDesMgr.pvItems[IDX_SERDES_ITEM].oSerCountOld == gPVSerDesMgr.pvItems[IDX_SERDES_ITEM].oSerCount)
		return;

	gPVSerDesMgr.pvItems[IDX_SERDES_ITEM].oSerCountOld = gPVSerDesMgr.pvItems[IDX_SERDES_ITEM].oSerCount;
	brsstrcpy((UDINT)txtMsg, (UDINT)"Pallet recipe saved to file.\n\nFilename: ");
	brsstrcat((UDINT)txtMsg, (UDINT)gPVSerDesMgr.pvItems[IDX_SERDES_ITEM].iFilename);
	paiHmiAlertShow(&gPaiHmiAlertMsg, "MESSAGE:", txtMsg, 3000);
}

void appHmiConfigFileCyclic(){

	if(gCtrl.main.btnLoadMachineCfg){//when hmi button pressed
		gCtrl.main.btnLoadMachineCfg = 0;
		appHmiAppConfigFileLoadRequest();//trigger AppConfig file load
	}

	if( gSerDesHMI_gConfigApp.oBtnClick ){
		gSerDesHMI_gConfigApp.oBtnClick = 0;
		paiHmiDialogShow(&gPaiHmiDialogMsg, "Application Configuration Is Changed!\n\nAccept and Save changes?", 10000, DLG_SaveAppConfigOK, DLG_SaveAppConfigCancel, 1);
	}

	if(gPaiHmiDialogMsg.result == DLG_SaveAppConfigOK){
		gPaiHmiDialogMsg.result = 0;
		appHmiAppConfigFileSaveRequest();
	}

	if(gPaiHmiDialogMsg.result == DLG_SaveAppConfigCancel){
		gPaiHmiDialogMsg.result = 0;
		appHmiAppConfigCancelChange();
	}

	appHmiAppConfigFileLoadEventCyclic();
	appHmiAppConfigFileSaveEventCyclic();
}

void appHmiPalletRecipeCyclic(){

	if( gSerDesHMI_gPalletCfg.oBtnClick ){
		gSerDesHMI_gPalletCfg.oBtnClick = 0;
		paiHmiDialogShow(&gPaiHmiDialogMsg, "Pallet Recipe Is Changed!\n\nAccept and Save changes?", 10000, DLG_SavePalletRecipeOK, DLG_SavePalletRecipeCancel, 1);
	}

	if(gPaiHmiDialogMsg.result == DLG_SavePalletRecipeOK){
		gPaiHmiDialogMsg.result = 0;
		appHmiPalletRecipeFileSaveRequest();
	}

	if(gPaiHmiDialogMsg.result == DLG_SavePalletRecipeCancel){
		gPaiHmiDialogMsg.result = 0;
		appHmiPalletRecipeCancelChange();
	}

	appHmiPalletRecipeFileSaveEventCyclic();
}

/*
###############################################################################
Init, Cyclic, Exit
###############################################################################
*/
void _INIT appHmiLogicInit(void)
{
	/* TODO: Add code here */

	paiRunningMsgInit(&gMsgRunningCtrl, gMsgRunning);
	gMsgRunningCtrl.iEnable = 1;
	gMsgRunningCtrl.iScrollDelayXms = 1000;
	gMsgRunningCtrl.iScrollLength = 100;

	//Remove
	gLayerEditorTxt.curIdxRow = 0;
	gLayerEditor.palCfgRows[0].palCfgCmds[0].cmdExtra = 0;

	//trigger cell selection on powerup
	gLayerEditorTxt.curIdxEditorCellOld = 1000;

	bgTimerStart(&gStats.runningTmr1sec, 1000);
	bgTimerStart(&gStats.runningTmr1min, 1000 * 60);
	bgTimerStart(&gStats.runningTmr1, 1000 * 60 * 60 * 24 * 100);

	//visibility flag for the pallet dispenser option
	gCtrl.palletDispenser.palletDispenserEquippedVis = gCtrl.palletDispenser.palletDispenserEquipped ? 0 : 1;

}
_LOCAL int gbTest;

//============================================================================
void _CYCLIC appHmiLogicCyclic(void)
{
	/* TODO: Add code here */

	//Logic to detect page change events and generate approprite signals / flags (i/e/ pageInit etc)
	paiHmiPageChangeCyclic(&gPaiHmiMain);

	//Page(screen) specific logic. Logic that runs/applies only to a specific page/screen
	screenHandlers(&gPaiHmiMain);

	if(gbTest == 1){
		gbTest = 0;
		// Show the alert with a specified text and for a selected amount of time
		paiHmiAlertShow(&gPaiHmiAlertMsg, "WARNING:","This is alert test!\nGoran Bjelcevic", 3000);
	}

	if(gbTest == 2){
		gbTest = 0;
		paiHmiDialogShow(&gPaiHmiDialogMsg, "Test or not?", 10000, 11, 12, 0);
	}

	if(gPaiHmiDialogMsg.result == 11){
		gPaiHmiDialogMsg.result = 0;
		paiHmiAlertShow(&gPaiHmiAlertMsg, "WARNING:", "Test 111.", 2000);
	}
	if(gPaiHmiDialogMsg.result == 12){
		gPaiHmiDialogMsg.result = 0;
		paiHmiAlertShow(&gPaiHmiAlertMsg, "WARNING:", "Test 222.", 2000);
	}

	paiRunningMsgCyclic(&gMsgRunningCtrl);
	if(gMsgRunningCtrl.curIdx < 30){
		gMsgRunningCtrl.oMsgFCIdx = 1;
	}else
	if(gMsgRunningCtrl.curIdx > 60){
		gMsgRunningCtrl.oMsgFCIdx = 2;
	}else{
		gMsgRunningCtrl.oMsgFCIdx = 0;
	}

	if(gCtrl.main.hmiShowMsgZeroingNeeded){
		gCtrl.main.hmiShowMsgZeroingNeeded = 0;
		paiHmiAlertShow(&gPaiHmiAlertMsg, "WARNING", "Machine Counts Changed!\nPlease Zero Machine!", 3000);
	}

	appHmiLayerEditor();

	appHmiPalleteEditorCyclic();

	appHmiLayerFileHandlerCyclic();
	appHmiPalleteFileHandlerCyclic();

	appHmiLayerL0L1FileLoadingCyclic();

	appScalingAndConversion();

	appBladeStopsUsed();

	appVisibilityCaseInfeedSide();

	appHmiConfigFileCyclic();

	appHmiPalletRecipeCyclic();

	appHmiGotoAlarmScreen();

}
//============================================================================
//EOF
```

### Program Logical/MachineControl/machmode
